KUKA KRL program: MyProgram_083().src

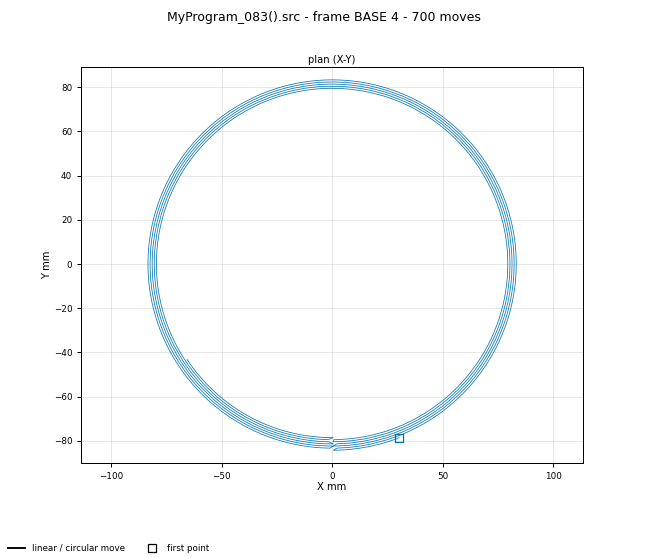
[picture p0: tool path of MyProgram_083().src in frame BASE 4, 700 of 700 moves have a stored position in this frame; points joined in program order, loops and branches not executed]
&ACCESS RVP
&REL 1
&PARAM TEMPLATE = C:\KRC\Roboter\Template\vorgabe
&PARAM EDITMASK = *
DEF MyProgram_083()
; ---- Setting reference (Base) ----
$BASE = BASE_DATA[4]

; --------------------------
; ---- Setting tool (TCP) ----
$TOOL = TOOL_DATA[3]
; --------------------------

$VEL.CP = VEL_APROX_PRINT
Startdeposition()
$VEL.CP = VEL_PRINT
LIN {X 30.3148,Y -78.5882,Z 83,A -74.2306,B 24.9241,C -2.0111,E1 25.0564,E2 519.1273} C_DIS
LIN {X 27.4017,Y -79.6507,Z 83,A -76.334,B 24.9244,C -2.0086,E1 25.0508,E2 521.2324} C_DIS
LIN {X 24.5836,Y -80.5643,Z 83,A -78.3586,B 24.9246,C -2.0059,E1 25.0454,E2 523.2596} C_DIS
LIN {X 21.4679,Y -81.4507,Z 83,A -80.5864,B 24.9248,C -2.0028,E1 25.0394,E2 525.4912} C_DIS
LIN {X 18.4554,Y -82.1857,Z 83,A -82.6471,B 24.9248,C -2.0023,E1 25.0338,E2 527.5502} C_DIS
LIN {X 15.4179,Y -82.8093,Z 83,A -84.7526,B 24.9249,C -2.0007,E1 25.028,E2 529.6571} C_DIS
LIN {X 12.3595,Y -83.3207,Z 83,A -86.9027,B 24.9252,C -1.9979,E1 25.0221,E2 531.8118} C_DIS
LIN {X 9.2843,Y -83.7191,Z 83,A -88.9651,B 24.9252,C -1.9981,E1 25.0164,E2 533.8722} C_DIS
LIN {X 6.1965,Y -84.0041,Z 83,A -91.0724,B 24.9252,C -1.9971,E1 25.0105,E2 535.9806} C_DIS
LIN {X 3.1004,Y -84.1753,Z 83,A -93.1799,B 24.9252,C -1.9963,E1 25.0046,E2 538.0892} C_DIS
LIN {X 0.5591,Y -84.2264,Z 83,A -94.1723,B 24.9236,C -2.0186,E1 25.002,E2 539.0288} C_DIS
Enddeposition()
LIN {X 0.5591,Y -84.2264,Z 83,A -94.1723,B 24.9236,C -2.0186,E1 25.002,E2 539.0288} C_DIS
Startdeposition()
$VEL.CP = VEL_PRINT
LIN {X 2.2766,Y -83.2483,Z 83,A -92.7209,B 24.9217,C -2.0436,E1 25.0063,E2 537.5182} C_DIS
LIN {X 5.5272,Y -83.0953,Z 83,A -90.5271,B 24.9217,C -2.0432,E1 25.0123,E2 535.3263} C_DIS
LIN {X 8.4362,Y -82.8508,Z 83,A -88.4909,B 24.9216,C -2.0451,E1 25.018,E2 533.2867} C_DIS
LIN {X 11.6914,Y -82.4542,Z 83,A -86.2486,B 24.9215,C -2.0461,E1 25.0242,E2 531.0439} C_DIS
LIN {X 14.5797,Y -81.9929,Z 83,A -84.2439,B 24.9214,C -2.0474,E1 25.0297,E2 529.0382} C_DIS
LIN {X 17.6429,Y -81.3887,Z 83,A -81.6481,B 24.9202,C -2.0634,E1 25.0369,E2 526.4078} C_DIS
LIN {X 24.7884,Y -79.5043,Z 83,A -76.0551,B 24.9185,C -2.0853,E1 25.052,E2 520.7724} C_DIS
LIN {X 29.127,Y -78.0202,Z 83,A -73.8096,B 24.9204,C -2.0602,E1 25.0578,E2 518.5911} C_DIS
LIN {X 32.2733,Y -76.7712,Z 83,A -71.5414,B 24.9204,C -2.0616,E1 25.0636,E2 516.3248} C_DIS
LIN {X 35.3444,Y -75.4069,Z 83,A -69.0733,B 24.9196,C -2.0701,E1 25.0699,E2 513.8426} C_DIS
LIN {X 38.5141,Y -73.8387,Z 83,A -66.2682,B 24.9184,C -2.0862,E1 25.077,E2 511.0072} C_DIS
LIN {X 41.3644,Y -72.2799,Z 83,A -64.0651,B 24.9181,C -2.0892,E1 25.0823,E2 508.8037} C_DIS
LIN {X 45.2001,Y -69.9456,Z 83,A -61.4311,B 24.9189,C -2.0802,E1 25.0885,E2 506.1994} C_DIS
LIN {X 47.8938,Y -68.1304,Z 83,A -59.266,B 24.9187,C -2.0823,E1 25.0934,E2 504.0366} C_DIS
LIN {X 50.4528,Y -66.258,Z 83,A -57.0629,B 24.9183,C -2.0876,E1 25.0984,E2 501.829} C_DIS
LIN {X 53.1162,Y -64.141,Z 83,A -54.8286,B 24.9181,C -2.0893,E1 25.1032,E2 499.5992} C_DIS
LIN {X 56.0538,Y -61.5911,Z 83,A -51.8123,B 24.9168,C -2.1066,E1 25.1096,E2 496.554} C_DIS
LIN {X 59.1004,Y -58.6733,Z 83,A -49.1949,B 24.917,C -2.1041,E1 25.1147,E2 493.9533} C_DIS
LIN {X 61.4699,Y -56.1859,Z 83,A -47.1294,B 24.9173,C -2.1002,E1 25.1186,E2 491.9062} C_DIS
LIN {X 64.0988,Y -53.1669,Z 83,A -44.0567,B 24.9159,C -2.1178,E1 25.1243,E2 488.8059} C_DIS
LIN {X 67.1499,Y -49.2572,Z 83,A -40.7875,B 24.9155,C -2.1221,E1 25.1298,E2 485.5419} C_DIS
LIN {X 68.7353,Y -47.0206,Z 83,A -38.365,B 24.9137,C -2.1453,E1 25.1337,E2 483.0767} C_DIS
LIN {X 71.2353,Y -43.1385,Z 83,A -35.7477,B 24.9145,C -2.1355,E1 25.1375,E2 480.4957} C_DIS
LIN {X 72.5407,Y -40.9065,Z 83,A -33.8555,B 24.9138,C -2.1444,E1 25.1402,E2 478.5923} C_DIS
LIN {X 74.1839,Y -37.8435,Z 83,A -31.5501,B 24.9134,C -2.1485,E1 25.1431,E2 476.2894} C_DIS
LIN {X 75.7192,Y -34.673,Z 83,A -29.1809,B 24.913,C -2.1539,E1 25.146,E2 473.9202} C_DIS
LIN {X 78.0639,Y -29.0114,Z 83,A -24.9527,B 24.9119,C -2.1671,E1 25.1504,E2 469.6842} C_DIS
LIN {X 79.3994,Y -25.1265,Z 83,A -22.1584,B 24.9113,C -2.1748,E1 25.1528,E2 466.8876} C_DIS
LIN {X 80.2886,Y -22.1198,Z 83,A -19.9737,B 24.9107,C -2.1825,E1 25.1545,E2 464.6972} C_DIS
LIN {X 81.1089,Y -18.8877,Z 83,A -17.759,B 24.9103,C -2.187,E1 25.156,E2 462.4846} C_DIS
LIN {X 81.8011,Y -15.6197,Z 83,A -15.3853,B 24.9095,C -2.1969,E1 25.1573,E2 460.1016} C_DIS
LIN {X 82.4143,Y -11.9722,Z 83,A -13.1383,B 24.9096,C -2.1949,E1 25.1583,E2 457.8722} C_DIS
LIN {X 82.7817,Y -9.0968,Z 83,A -10.9181,B 24.9085,C -2.2089,E1 25.159,E2 455.6322} C_DIS
LIN {X 83.0508,Y -6.1767,Z 83,A -9.0557,B 24.9084,C -2.2101,E1 25.1594,E2 453.778} C_DIS
LIN {X 83.1967,Y -3.7006,Z 83,A -7.1515,B 24.9074,C -2.2223,E1 25.1597,E2 451.8564} C_DIS
LIN {X 83.2798,Y 0.1338,Z 83,A -4.6895,B 24.9072,C -2.2247,E1 25.1597,E2 449.4032} C_DIS
LIN {X 83.2317,Y 2.8163,Z 83,A -2.9547,B 24.907,C -2.2269,E1 25.1597,E2 447.6737} C_DIS
LIN {X 83.0758,Y 5.8158,Z 83,A -0.6903,B 24.9059,C -2.2401,E1 25.1593,E2 445.3915} C_DIS
LIN {X 82.796,Y 8.96,Z 83,A 1.5055,B 24.9052,C -2.2477,E1 25.1586,E2 443.1907} C_DIS
LIN {X 82.3293,Y 12.5416,Z 83,A 3.8863,B 24.9049,C -2.252,E1 25.1577,E2 440.8138} C_DIS
LIN {X 81.7324,Y 15.9765,Z 83,A 6.3167,B 24.9041,C -2.2605,E1 25.1565,E2 438.3776} C_DIS
LIN {X 81.047,Y 19.1557,Z 83,A 8.3166,B 24.9042,C -2.2594,E1 25.1553,E2 436.3919} C_DIS
LIN {X 79.9547,Y 23.2977,Z 83,A 11.4453,B 24.903,C -2.2744,E1 25.153,E2 433.2459} C_DIS
LIN {X 78.9726,Y 26.4336,Z 83,A 13.6144,B 24.9026,C -2.278,E1 25.1511,E2 431.0804} C_DIS
LIN {X 78.1039,Y 28.9017,Z 83,A 15.9195,B 24.9007,C -2.3002,E1 25.1488,E2 428.7359} C_DIS
LIN {X 76.3834,Y 33.1808,Z 83,A 18.5771,B 24.9014,C -2.2921,E1 25.146,E2 426.112} C_DIS
LIN {X 74.9893,Y 36.2217,Z 83,A 20.8163,B 24.9011,C -2.2964,E1 25.1433,E2 423.8746} C_DIS
LIN {X 73.5484,Y 39.0652,Z 83,A 23.1175,B 24.9002,C -2.306,E1 25.1404,E2 421.563} C_DIS
LIN {X 72.3086,Y 41.3145,Z 83,A 24.9996,B 24.8995,C -2.3145,E1 25.1378,E2 419.6705} C_DIS
LIN {X 70.4163,Y 44.4645,Z 83,A 27.2243,B 24.8998,C -2.3111,E1 25.1345,E2 417.4651} C_DIS
LIN {X 68.659,Y 47.1334,Z 83,A 29.3239,B 24.8996,C -2.3134,E1 25.1313,E2 415.3705} C_DIS
LIN {X 66.949,Y 49.5316,Z 83,A 31.5565,B 24.8986,C -2.3252,E1 25.1276,E2 413.121} C_DIS
LIN {X 65.0896,Y 51.9507,Z 83,A 33.6147,B 24.8982,C -2.3288,E1 25.124,E2 411.0638} C_DIS
LIN {X 63.2176,Y 54.2123,Z 83,A 35.6181,B 24.8979,C -2.333,E1 25.1204,E2 409.0597} C_DIS
LIN {X 60.497,Y 57.2324,Z 83,A 38.4466,B 24.8972,C -2.3402,E1 25.1151,E2 406.2267} C_DIS
LIN {X 58.1763,Y 59.5914,Z 83,A 40.7466,B 24.8968,C -2.3457,E1 25.1105,E2 403.9233} C_DIS
LIN {X 56.3761,Y 61.2954,Z 83,A 42.6082,B 24.896,C -2.3542,E1 25.1067,E2 402.0492} C_DIS
LIN {X 53.5749,Y 63.7598,Z 83,A 45.0221,B 24.896,C -2.3542,E1 25.1016,E2 399.6447} C_DIS
LIN {X 50.8443,Y 65.9563,Z 83,A 47.0753,B 24.8966,C -2.3472,E1 25.0971,E2 397.6158} C_DIS
LIN {X 48.675,Y 67.5741,Z 83,A 49.1394,B 24.8958,C -2.3568,E1 25.0925,E2 395.5362} C_DIS
LIN {X 46.1454,Y 69.3261,Z 83,A 51.7586,B 24.894,C -2.3762,E1 25.0863,E2 392.8798} C_DIS
LIN {X 41.7622,Y 72.0513,Z 83,A 54.8615,B 24.8948,C -2.3672,E1 25.079,E2 389.8078} C_DIS
LIN {X 38.8786,Y 73.6467,Z 83,A 57.1378,B 24.8945,C -2.3706,E1 25.0734,E2 387.5302} C_DIS
LIN {X 35.9344,Y 75.1273,Z 83,A 59.3109,B 24.8945,C -2.3704,E1 25.0679,E2 385.3633} C_DIS
LIN {X 33.2525,Y 76.3521,Z 83,A 61.146,B 24.8949,C -2.3666,E1 25.0633,E2 383.5416} C_DIS
LIN {X 29.1509,Y 78.0111,Z 83,A 64.9693,B 24.8925,C -2.3939,E1 25.0532,E2 379.6623} C_DIS
LIN {X 26.0378,Y 79.1049,Z 83,A 66.6073,B 24.8941,C -2.3761,E1 25.049,E2 378.0695} C_DIS
LIN {X 24.074,Y 79.7244,Z 83,A 68.1871,B 24.8935,C -2.3822,E1 25.0447,E2 376.4781} C_DIS
LIN {X 20.7113,Y 80.6624,Z 83,A 70.3301,B 24.8941,C -2.3758,E1 25.039,E2 374.3537} C_DIS
LIN {X 18.1998,Y 81.2672,Z 83,A 72.3695,B 24.8933,C -2.3847,E1 25.0334,E2 372.2959} C_DIS
LIN {X 14.9781,Y 81.9212,Z 83,A 74.5372,B 24.8935,C -2.3828,E1 25.0275,E2 370.1353} C_DIS
LIN {X 12.2266,Y 82.3779,Z 83,A 76.2737,B 24.8939,C -2.3778,E1 25.0227,E2 368.4123} C_DIS
LIN {X 9.7923,Y 82.7013,Z 83,A 78.135,B 24.8934,C -2.3834,E1 25.0175,E2 366.5393} C_DIS
LIN {X 6.4728,Y 83.0271,Z 83,A 80.4499,B 24.8934,C -2.3842,E1 25.0111,E2 364.2238} C_DIS
LIN {X 3.2103,Y 83.2178,Z 83,A 82.8056,B 24.8931,C -2.3873,E1 25.0045,E2 361.8615} C_DIS
LIN {X -0.433,Y 83.2778,Z 83,A 85.1471,B 24.8935,C -2.3819,E1 24.998,E2 359.5329} C_DIS
LIN {X -3.6284,Y 83.1998,Z 83,A 87.3137,B 24.8937,C -2.3803,E1 24.992,E2 357.3698} C_DIS
LIN {X -6.4631,Y 83.0279,Z 83,A 89.3062,B 24.8937,C -2.3806,E1 24.9864,E2 355.3758} C_DIS
LIN {X -10.1051,Y 82.6646,Z 83,A 91.8731,B 24.8937,C -2.3806,E1 24.9793,E2 352.8072} C_DIS
LIN {X -13.5154,Y 82.1752,Z 83,A 94.2123,B 24.8939,C -2.3782,E1 24.9728,E2 350.4719} C_DIS
LIN {X -16.3634,Y 81.6564,Z 83,A 96.287,B 24.8938,C -2.379,E1 24.9671,E2 348.3929} C_DIS
LIN {X -19.702,Y 80.9148,Z 83,A 98.5118,B 24.8943,C -2.3732,E1 24.9611,E2 346.1791} C_DIS
LIN {X -22.4154,Y 80.2061,Z 83,A 100.4183,B 24.8946,C -2.3705,E1 24.956,E2 344.2759} C_DIS
LIN {X -24.918,Y 79.4641,Z 83,A 102.3404,B 24.8944,C -2.3722,E1 24.9508,E2 342.3467} C_DIS
LIN {X -27.7638,Y 78.5149,Z 83,A 104.7794,B 24.8937,C -2.3804,E1 24.9443,E2 339.8832} C_DIS
LIN {X -31.8944,Y 76.9307,Z 83,A 107.4713,B 24.8949,C -2.3662,E1 24.9374,E2 337.2195} C_DIS
LIN {X -34.8305,Y 75.6461,Z 83,A 109.7266,B 24.8951,C -2.3643,E1 24.9317,E2 334.963} C_DIS
LIN {X -41.0642,Y 72.4518,Z 83,A 114.2822,B 24.8965,C -2.3489,E1 24.9205,E2 330.4317} C_DIS
LIN {X -43.5772,Y 70.9687,Z 83,A 116.6283,B 24.896,C -2.3548,E1 24.9148,E2 328.0644} C_DIS
LIN {X -46.1606,Y 69.3161,Z 83,A 118.8803,B 24.896,C -2.3548,E1 24.9095,E2 325.8051} C_DIS
LIN {X -49.3998,Y 67.0455,Z 83,A 121.4238,B 24.8969,C -2.3442,E1 24.9038,E2 323.2778} C_DIS
LIN {X -52.0211,Y 65.0339,Z 83,A 123.4956,B 24.8978,C -2.3338,E1 24.8993,E2 321.2231} C_DIS
LIN {X -54.4202,Y 63.04,Z 83,A 126.0988,B 24.8971,C -2.3417,E1 24.8937,E2 318.591} C_DIS
LIN {X -57.2714,Y 60.4604,Z 83,A 128.4357,B 24.8984,C -2.3271,E1 24.8889,E2 316.2794} C_DIS
LIN {X -59.3395,Y 58.4313,Z 83,A 130.5413,B 24.8985,C -2.3254,E1 24.8848,E2 314.169} C_DIS
LIN {X -61.8347,Y 55.7848,Z 83,A 132.9601,B 24.8993,C -2.3169,E1 24.8802,E2 311.7598} C_DIS
LIN {X -64.2217,Y 53.0191,Z 83,A 135.5053,B 24.8998,C -2.3114,E1 24.8756,E2 309.2162} C_DIS
LIN {X -66.1385,Y 50.6079,Z 83,A 137.4999,B 24.9005,C -2.3024,E1 24.8722,E2 307.2336} C_DIS
LIN {X -68.0525,Y 48.0045,Z 83,A 139.9954,B 24.9005,C -2.3038,E1 24.8681,E2 304.7225} C_DIS
LIN {X -71.4518,Y 42.7801,Z 83,A 143.9677,B 24.9022,C -2.2832,E1 24.8622,E2 300.7793} C_DIS
LIN {X -73.1359,Y 39.8313,Z 83,A 146.5293,B 24.9022,C -2.2826,E1 24.8587,E2 298.2058} C_DIS
LIN {X -74.6288,Y 36.9583,Z 83,A 148.8382,B 24.9026,C -2.2783,E1 24.8558,E2 295.8948} C_DIS
LIN {X -76.0363,Y 33.9695,Z 83,A 151.2402,B 24.9029,C -2.275,E1 24.853,E2 293.4876} C_DIS
LIN {X -77.4282,Y 30.6645,Z 83,A 153.607,B 24.9038,C -2.2648,E1 24.8505,E2 291.1318} C_DIS
LIN {X -78.3743,Y 28.1604,Z 83,A 155.2561,B 24.9047,C -2.254,E1 24.8489,E2 289.4992} C_DIS
LIN {X -79.7646,Y 23.9384,Z 83,A 158.5508,B 24.905,C -2.2508,E1 24.8461,E2 286.1931} C_DIS
LIN {X -80.7118,Y 20.5192,Z 83,A 160.9934,B 24.9056,C -2.2432,E1 24.8443,E2 283.7545} C_DIS
LIN {X -81.2535,Y 18.2619,Z 83,A 163.0357,B 24.905,C -2.2502,E1 24.8431,E2 281.6836} C_DIS
LIN {X -82.1577,Y 13.62,Z 83,A 165.639,B 24.9074,C -2.2224,E1 24.8418,E2 279.1312} C_DIS
LIN {X -82.6677,Y 10.0792,Z 83,A 168.3253,B 24.9075,C -2.2206,E1 24.8408,E2 276.4333} C_DIS
LIN {X -82.9964,Y 6.8574,Z 83,A 170.4206,B 24.9084,C -2.2099,E1 24.8402,E2 274.3509} C_DIS
LIN {X -83.1884,Y 3.8947,Z 83,A 172.6479,B 24.9085,C -2.2083,E1 24.8399,E2 272.1139} C_DIS
LIN {X -83.2762,Y 0.7426,Z 83,A 174.7922,B 24.9092,C -2.2007,E1 24.8398,E2 269.9748} C_DIS
LIN {X -83.2493,Y -2.2433,Z 83,A 176.8695,B 24.9096,C -2.1948,E1 24.8398,E2 267.8991} C_DIS
LIN {X -83.1174,Y -5.2015,Z 83,A 178.9156,B 24.9102,C -2.1886,E1 24.8402,E2 265.8556} C_DIS
LIN {X -82.869,Y -8.263,Z 83,A -178.9161,B 24.9106,C -2.1834,E1 24.8407,E2 263.6867} C_DIS
LIN {X -82.5154,Y -11.2599,Z 83,A -176.8353,B 24.9111,C -2.177,E1 24.8415,E2 261.6086} C_DIS
LIN {X -82.0089,Y -14.491,Z 83,A -174.0318,B 24.9104,C -2.1851,E1 24.8428,E2 258.7694} C_DIS
LIN {X -81.3812,Y -17.6772,Z 83,A -172.376,B 24.9123,C -2.1625,E1 24.8438,E2 257.1577} C_DIS
LIN {X -80.806,Y -20.148,Z 83,A -170.2993,B 24.912,C -2.1661,E1 24.8452,E2 255.0601} C_DIS
LIN {X -79.7539,Y -23.9746,Z 83,A -167.8923,B 24.9134,C -2.1492,E1 24.847,E2 252.6797} C_DIS
LIN {X -78.8305,Y -26.8552,Z 83,A -165.8053,B 24.9139,C -2.1432,E1 24.8488,E2 250.5951} C_DIS
LIN {X -77.9352,Y -29.3513,Z 83,A -163.8576,B 24.914,C -2.1412,E1 24.8507,E2 248.641} C_DIS
LIN {X -76.8139,Y -32.172,Z 83,A -161.7124,B 24.9144,C -2.1368,E1 24.853,E2 246.4945} C_DIS
LIN {X -75.485,Y -35.1767,Z 83,A -159.5329,B 24.9151,C -2.1282,E1 24.8555,E2 244.3234} C_DIS
LIN {X -73.9824,Y -38.2378,Z 83,A -157.1587,B 24.9155,C -2.1225,E1 24.8585,E2 241.9501} C_DIS
LIN {X -72.4839,Y -41.0083,Z 83,A -154.8521,B 24.9157,C -2.1206,E1 24.8616,E2 239.6361} C_DIS
LIN {X -70.6438,Y -44.1002,Z 83,A -152.5429,B 24.9165,C -2.1095,E1 24.8649,E2 237.3413} C_DIS
LIN {X -69.2182,Y -46.3077,Z 83,A -150.0661,B 24.9154,C -2.1235,E1 24.8689,E2 234.8187} C_DIS
LIN {X -67.277,Y -49.0836,Z 83,A -148.293,B 24.9171,C -2.1023,E1 24.8717,E2 233.0878} C_DIS
LIN {X -65.2096,Y -51.7989,Z 83,A -146.2559,B 24.9182,C -2.088,E1 24.8751,E2 231.075} C_DIS
LIN {X -63.0232,Y -54.4395,Z 83,A -143.4942,B 24.9178,C -2.0938,E1 24.8801,E2 228.2867} C_DIS
LIN {X -60.8121,Y -56.8974,Z 83,A -141.3418,B 24.9184,C -2.0854,E1 24.8842,E2 226.1449} C_DIS
LIN {X -58.9873,Y -58.7879,Z 83,A -138.93,B 24.9174,C -2.0987,E1 24.889,E2 223.6911} C_DIS
LIN {X -56.6005,Y -61.0895,Z 83,A -137.1338,B 24.9188,C -2.0803,E1 24.8926,E2 221.9315} C_DIS
LIN {X -54.085,Y -63.3261,Z 83,A -134.6178,B 24.9188,C -2.0816,E1 24.8979,E2 219.4026} C_DIS
LIN {X -50.8394,Y -65.9601,Z 83,A -131.9262,B 24.9196,C -2.0711,E1 24.9038,E2 216.726} C_DIS
LIN {X -48.6875,Y -67.5652,Z 83,A -129.5874,B 24.9187,C -2.0821,E1 24.9092,E2 214.3527} C_DIS
LIN {X -46.0328,Y -69.4004,Z 83,A -127.8872,B 24.9201,C -2.0636,E1 24.913,E2 212.691} C_DIS
LIN {X -42.9611,Y -71.3431,Z 83,A -125.3297,B 24.9203,C -2.0615,E1 24.9191,E2 210.1304} C_DIS
LIN {X -40.114,Y -72.9826,Z 83,A -123.2403,B 24.9209,C -2.0535,E1 24.9242,E2 208.0541} C_DIS
LIN {X -37.7618,Y -74.2256,Z 83,A -121.4189,B 24.9211,C -2.0509,E1 24.9287,E2 206.2338} C_DIS
LIN {X -35.3141,Y -75.421,Z 83,A -118.7338,B 24.9194,C -2.0726,E1 24.9356,E2 203.4904} C_DIS
LIN {X -31.9021,Y -76.9276,Z 83,A -116.0869,B 24.9194,C -2.0724,E1 24.9424,E2 200.838} C_DIS
LIN {X -28.2936,Y -78.3257,Z 83,A -114.32,B 24.9217,C -2.0434,E1 24.9469,E2 199.1363} C_DIS
LIN {X -25.3736,Y -79.3198,Z 83,A -111.9912,B 24.9214,C -2.0479,E1 24.9531,E2 196.7926} C_DIS
LIN {X -22.809,Y -80.0946,Z 83,A -110.2382,B 24.9217,C -2.044,E1 24.9578,E2 195.0461} C_DIS
LIN {X -19.6726,Y -80.922,Z 83,A -107.9499,B 24.9217,C -2.0444,E1 24.964,E2 192.7535} C_DIS
LIN {X -16.8864,Y -81.5491,Z 83,A -106.0101,B 24.9217,C -2.0428,E1 24.9693,E2 190.8152} C_DIS
LIN {X -13.5662,Y -82.1667,Z 83,A -103.7836,B 24.922,C -2.0391,E1 24.9754,E2 188.5951} C_DIS
LIN {X -10.5031,Y -82.6142,Z 83,A -101.4942,B 24.9217,C -2.0435,E1 24.9818,E2 186.2935} C_DIS
LIN {X -7.1182,Y -82.9756,Z 83,A -99.121,B 24.9217,C -2.0442,E1 24.9884,E2 183.9173} C_DIS
LIN {X -4.5308,Y -83.1556,Z 83,A -97.373,B 24.9217,C -2.0432,E1 24.9932,E2 182.1712} C_DIS
LIN {X -1.0027,Y -83.2741,Z 83,A -94.9241,B 24.9217,C -2.0442,E1 25.0001,E2 179.7197} C_DIS
LIN {X -1.0027,Y -83.2741,Z 83,A -94.9241,B 24.9217,C -2.0442,E1 25.0001,E2 179.7197} C_DIS
Enddeposition()
LIN {X 0.5504,Y -82.3231,Z 83,A -94.2468,B 24.9213,C -2.049,E1 25.002,E2 179.031} C_DIS
Startdeposition()
$VEL.CP = VEL_PRINT
LIN {X -1.5524,Y -82.3124,Z 83,A -96.6682,B 24.9235,C -2.0201,E1 24.9951,E2 181.5212} C_DIS
LIN {X -5.6861,Y -82.1306,Z 83,A -99.1832,B 24.9227,C -2.0307,E1 24.9881,E2 184.0117} C_DIS
LIN {X -8.7147,Y -81.8646,Z 83,A -101.4384,B 24.923,C -2.0267,E1 24.9818,E2 186.2775} C_DIS
LIN {X -11.9249,Y -81.4596,Z 83,A -103.7765,B 24.9231,C -2.0247,E1 24.9753,E2 188.6223} C_DIS
LIN {X -15.5144,Y -80.852,Z 83,A -106.1545,B 24.9227,C -2.0301,E1 24.9688,E2 190.99} C_DIS
LIN {X -18.5189,Y -80.2172,Z 83,A -108.3547,B 24.9227,C -2.0292,E1 24.9628,E2 193.1948} C_DIS
LIN {X -22.5796,Y -79.1702,Z 83,A -110.9842,B 24.922,C -2.0393,E1 24.9558,E2 195.8044} C_DIS
LIN {X -24.8256,Y -78.4957,Z 83,A -113.2233,B 24.9233,C -2.023,E1 24.9497,E2 198.086} C_DIS
LIN {X -28.7698,Y -77.1376,Z 83,A -116.3221,B 24.9235,C -2.02,E1 24.9415,E2 201.1981} C_DIS
LIN {X -34.6143,Y -74.6968,Z 83,A -120.2039,B 24.922,C -2.0396,E1 24.9317,E2 205.0426} C_DIS
LIN {X -37.6746,Y -73.2013,Z 83,A -122.7566,B 24.9222,C -2.0374,E1 24.9253,E2 207.6075} C_DIS
LIN {X -40.8894,Y -71.455,Z 83,A -125.1525,B 24.9216,C -2.045,E1 24.9194,E2 209.992} C_DIS
LIN {X -43.7124,Y -69.7638,Z 83,A -127.7428,B 24.922,C -2.0401,E1 24.9132,E2 212.6022} C_DIS
LIN {X -48.0318,Y -66.8637,Z 83,A -131.0831,B 24.9209,C -2.0537,E1 24.9056,E2 215.9213} C_DIS
LIN {X -50.4597,Y -65.051,Z 83,A -133.24,B 24.9207,C -2.0561,E1 24.9008,E2 218.0804} C_DIS
LIN {X -53.9999,Y -62.1434,Z 83,A -136.1063,B 24.9196,C -2.0709,E1 24.8947,E2 220.9224} C_DIS
LIN {X -56.6894,Y -59.701,Z 83,A -139.5018,B 24.921,C -2.0523,E1 24.8876,E2 224.3759} C_DIS
LIN {X -58.9888,Y -57.4303,Z 83,A -141.2543,B 24.9196,C -2.0705,E1 24.8843,E2 226.0926} C_DIS
LIN {X -61.1234,Y -55.1523,Z 83,A -144.227,B 24.9209,C -2.0538,E1 24.8786,E2 229.1183} C_DIS
LIN {X -63.782,Y -52.0545,Z 83,A -146.3247,B 24.9188,C -2.0802,E1 24.875,E2 231.1626} C_DIS
LIN {X -66.5611,Y -48.4501,Z 83,A -149.7864,B 24.9188,C -2.08,E1 24.8691,E2 234.6415} C_DIS
LIN {X -69.0207,Y -44.879,Z 83,A -152.4967,B 24.9176,C -2.0958,E1 24.865,E2 237.3277} C_DIS
LIN {X -70.5517,Y -42.4305,Z 83,A -155.1104,B 24.9185,C -2.0851,E1 24.8611,E2 239.9804} C_DIS
LIN {X -72.2473,Y -39.4733,Z 83,A -156.9169,B 24.9168,C -2.1064,E1 24.8587,E2 241.7455} C_DIS
LIN {X -73.8018,Y -36.4834,Z 83,A -159.2444,B 24.9162,C -2.1133,E1 24.8558,E2 244.0691} C_DIS
LIN {X -75.8072,Y -32.1097,Z 83,A -162.5765,B 24.9155,C -2.1231,E1 24.852,E2 247.3959} C_DIS
LIN {X -76.9221,Y -29.3391,Z 83,A -164.668,B 24.915,C -2.1288,E1 24.8499,E2 249.4857} C_DIS
LIN {X -77.9197,Y -26.5773,Z 83,A -166.7483,B 24.9146,C -2.1338,E1 24.8479,E2 251.5658} C_DIS
LIN {X -78.9025,Y -23.4978,Z 83,A -169.0526,B 24.9142,C -2.1391,E1 24.846,E2 253.8707} C_DIS
LIN {X -80.1273,Y -18.9078,Z 83,A -172.4738,B 24.9136,C -2.1461,E1 24.8437,E2 257.2951} C_DIS
LIN {X -81.1733,Y -13.7358,Z 83,A -175.6492,B 24.9116,C -2.1704,E1 24.842,E2 260.4312} C_DIS
LIN {X -81.5066,Y -11.594,Z 83,A -177.5733,B 24.9121,C -2.1643,E1 24.8412,E2 262.3815} C_DIS
LIN {X -82.0324,Y -6.972,Z 83,A 178.7589,B 24.9122,C -2.1633,E1 24.8402,E2 266.0735} C_DIS
LIN {X -82.2721,Y -3.0466,Z 83,A 176.3153,B 24.9109,C -2.1796,E1 24.8398,E2 268.4931} C_DIS
LIN {X -82.3268,Y 0.3626,Z 83,A 173.6639,B 24.9109,C -2.18,E1 24.8398,E2 271.1595} C_DIS
LIN {X -82.0421,Y 6.8502,Z 83,A 169.7779,B 24.9083,C -2.2108,E1 24.8404,E2 274.9953} C_DIS
LIN {X -81.6591,Y 10.4669,Z 83,A 166.5866,B 24.9091,C -2.2018,E1 24.8414,E2 278.2273} C_DIS
LIN {X -81.2236,Y 13.4345,Z 83,A 164.049,B 24.9095,C -2.1968,E1 24.8426,E2 280.7917} C_DIS
LIN {X -80.5008,Y 17.243,Z 83,A 162.0067,B 24.9074,C -2.2222,E1 24.8437,E2 282.7855} C_DIS
LIN {X -79.9755,Y 19.5361,Z 83,A 159.576,B 24.9086,C -2.207,E1 24.8454,E2 285.2667} C_DIS
LIN {X -78.8665,Y 23.6193,Z 83,A 157.1283,B 24.9068,C -2.2288,E1 24.8473,E2 287.6764} C_DIS
LIN {X -77.4401,Y 27.9437,Z 83,A 154.6172,B 24.9046,C -2.2557,E1 24.8495,E2 290.1378} C_DIS
LIN {X -76.529,Y 30.3501,Z 83,A 152.4182,B 24.905,C -2.2505,E1 24.8517,E2 292.3615} C_DIS
LIN {X -74.1199,Y 35.8333,Z 83,A 148.4322,B 24.9035,C -2.2677,E1 24.8563,E2 296.3283} C_DIS
LIN {X -71.2191,Y 41.3001,Z 83,A 144.1422,B 24.9024,C -2.2806,E1 24.862,E2 300.6102} C_DIS
LIN {X -70.2138,Y 42.9864,Z 83,A 141.9782,B 24.9039,C -2.2636,E1 24.8652,E2 302.8258} C_DIS
LIN {X -68.3701,Y 45.8628,Z 83,A 140.1448,B 24.9021,C -2.2844,E1 24.868,E2 304.6189} C_DIS
LIN {X -65.4603,Y 49.9285,Z 83,A 136.7915,B 24.901,C -2.297,E1 24.8735,E2 307.9581} C_DIS
LIN {X -62.0296,Y 54.1301,Z 83,A 133.0235,B 24.9001,C -2.3069,E1 24.8802,E2 311.7199} C_DIS
LIN {X -59.2782,Y 57.13,Z 83,A 130.55,B 24.8987,C -2.3235,E1 24.8848,E2 314.1648} C_DIS
LIN {X -57.8082,Y 58.617,Z 83,A 128.5469,B 24.8997,C -2.3124,E1 24.8888,E2 316.2029} C_DIS
LIN {X -54.1458,Y 62.016,Z 83,A 125.3768,B 24.8983,C -2.3286,E1 24.8953,E2 319.3472} C_DIS
LIN {X -50.9579,Y 64.6611,Z 83,A 122.3567,B 24.898,C -2.3311,E1 24.9018,E2 322.3727} C_DIS
LIN {X -48.8772,Y 66.2484,Z 83,A 119.525,B 24.9001,C -2.3078,E1 24.9083,E2 325.2699} C_DIS
LIN {X -45.5242,Y 68.5956,Z 83,A 117.8431,B 24.8968,C -2.3447,E1 24.912,E2 326.8695} C_DIS
LIN {X -42.0842,Y 70.7581,Z 83,A 114.7218,B 24.8971,C -2.342,E1 24.9194,E2 330.0073} C_DIS
LIN {X -38.4333,Y 72.8054,Z 83,A 111.4114,B 24.8976,C -2.3361,E1 24.9276,E2 333.3411} C_DIS
LIN {X -35.4537,Y 74.3023,Z 83,A 109.3633,B 24.8966,C -2.3472,E1 24.9327,E2 335.368} C_DIS
LIN {X -32.558,Y 75.6165,Z 83,A 107.135,B 24.8964,C -2.35,E1 24.9384,E2 337.595} C_DIS
LIN {X -27.5644,Y 77.5761,Z 83,A 103.429,B 24.8959,C -2.3557,E1 24.948,E2 341.2953} C_DIS
LIN {X -23.8211,Y 78.8061,Z 83,A 100.2076,B 24.8968,C -2.3455,E1 24.9567,E2 344.5465} C_DIS
LIN {X -19.399,Y 80.009,Z 83,A 97.4156,B 24.8955,C -2.3597,E1 24.9642,E2 347.3088} C_DIS
LIN {X -16.0884,Y 80.7412,Z 83,A 94.203,B 24.8975,C -2.3378,E1 24.9731,E2 350.5772} C_DIS
LIN {X -11.8028,Y 81.4769,Z 83,A 92.347,B 24.8943,C -2.3728,E1 24.978,E2 352.3515} C_DIS
LIN {X -7.1632,Y 82.0158,Z 83,A 89.0161,B 24.8943,C -2.3723,E1 24.9873,E2 355.6859} C_DIS
LIN {X -4.347,Y 82.2124,Z 83,A 86.8115,B 24.8949,C -2.3662,E1 24.9935,E2 357.9058} C_DIS
LIN {X 0.5328,Y 82.3253,Z 83,A 83.2747,B 24.8952,C -2.3629,E1 25.0034,E2 361.4503} C_DIS
LIN {X 3.3202,Y 82.2604,Z 83,A 81.4837,B 24.8948,C -2.3674,E1 25.0083,E2 363.2303} C_DIS
LIN {X 6.5866,Y 82.0632,Z 83,A 79.2593,B 24.8947,C -2.3689,E1 25.0145,E2 365.4501} C_DIS
LIN {X 10.5225,Y 81.6518,Z 83,A 76.3504,B 24.8951,C -2.3639,E1 25.0226,E2 368.3687} C_DIS
LIN {X 13.7049,Y 81.1784,Z 83,A 74.1891,B 24.8951,C -2.3655,E1 25.0285,E2 370.5241} C_DIS
LIN {X 16.9177,Y 80.5709,Z 83,A 71.5231,B 24.8961,C -2.353,E1 25.0359,E2 373.2164} C_DIS
LIN {X 21.5203,Y 79.4646,Z 83,A 68.4024,B 24.8958,C -2.3561,E1 25.0443,E2 376.325} C_DIS
LIN {X 25.4418,Y 78.2973,Z 83,A 65.6913,B 24.8957,C -2.358,E1 25.0515,E2 379.0266} C_DIS
LIN {X 31.7462,Y 75.9604,Z 83,A 61.5346,B 24.8947,C -2.3693,E1 25.0623,E2 383.1475} C_DIS
LIN {X 36.255,Y 73.9151,Z 83,A 57.8652,B 24.8956,C -2.3585,E1 25.0716,E2 386.8333} C_DIS
LIN {X 38.8943,Y 72.5613,Z 83,A 55.6569,B 24.8962,C -2.3515,E1 25.0771,E2 389.0522} C_DIS
LIN {X 41.8717,Y 70.8837,Z 83,A 53.2243,B 24.8967,C -2.3464,E1 25.083,E2 391.4893} C_DIS
LIN {X 45.4938,Y 68.6156,Z 83,A 50.5294,B 24.8963,C -2.3504,E1 25.0893,E2 394.166} C_DIS
LIN {X 47.6472,Y 67.1382,Z 83,A 47.8331,B 24.899,C -2.3204,E1 25.0956,E2 396.9242} C_DIS
LIN {X 50.6928,Y 64.8706,Z 83,A 45.9418,B 24.8974,C -2.3388,E1 25.0997,E2 398.765} C_DIS
LIN {X 53.0351,Y 62.9701,Z 83,A 42.9527,B 24.9001,C -2.3073,E1 25.1062,E2 401.817} C_DIS
LIN {X 56.1846,Y 60.1757,Z 83,A 40.9125,B 24.8982,C -2.329,E1 25.1103,E2 403.7975} C_DIS
LIN {X 58.4013,Y 58.0266,Z 83,A 38.7825,B 24.8986,C -2.3251,E1 25.1145,E2 405.9279} C_DIS
LIN {X 61.9206,Y 54.255,Z 83,A 35.2623,B 24.8991,C -2.3194,E1 25.1212,E2 409.4461} C_DIS
LIN {X 63.8799,Y 51.9337,Z 83,A 33.0856,B 24.8997,C -2.3125,E1 25.125,E2 411.6291} C_DIS
LIN {X 67.3106,Y 47.4055,Z 83,A 29.1432,B 24.9005,C -2.3032,E1 25.1316,E2 415.5746} C_DIS
LIN {X 69.64,Y 43.9105,Z 83,A 25.5133,B 24.903,C -2.2733,E1 25.1372,E2 419.2569} C_DIS
LIN {X 71.6242,Y 40.595,Z 83,A 23.5565,B 24.9017,C -2.2894,E1 25.1398,E2 421.1655} C_DIS
LIN {X 73.1055,Y 37.862,Z 83,A 21.3371,B 24.9023,C -2.2817,E1 25.1427,E2 423.3914} C_DIS
LIN {X 74.8291,Y 34.33,Z 83,A 18.785,B 24.9025,C -2.28,E1 25.1458,E2 425.9339} C_DIS
LIN {X 76.0477,Y 31.539,Z 83,A 16.0179,B 24.9048,C -2.2531,E1 25.1488,E2 428.7492} C_DIS
LIN {X 77.2546,Y 28.4522,Z 83,A 13.9451,B 24.9048,C -2.2539,E1 25.1508,E2 430.8086} C_DIS
LIN {X 78.349,Y 25.2821,Z 83,A 10.7448,B 24.9076,C -2.2192,E1 25.1536,E2 434.0725} C_DIS
LIN {X 79.8503,Y 20.047,Z 83,A 8.4245,B 24.9046,C -2.255,E1 25.1552,E2 436.2951} C_DIS
LIN {X 80.4835,Y 17.3262,Z 83,A 6.3022,B 24.9056,C -2.2433,E1 25.1565,E2 438.4328} C_DIS
LIN {X 81.0354,Y 14.5263,Z 83,A 4.3727,B 24.906,C -2.239,E1 25.1575,E2 440.3611} C_DIS
LIN {X 81.5472,Y 11.3083,Z 83,A 1.9681,B 24.9069,C -2.2274,E1 25.1585,E2 442.7788} C_DIS
LIN {X 81.935,Y 8.0372,Z 83,A -0.0012,B 24.9067,C -2.2307,E1 25.1591,E2 444.7286} C_DIS
LIN {X 82.1268,Y 5.7416,Z 83,A -1.7324,B 24.9074,C -2.2215,E1 25.1595,E2 446.4714} C_DIS
LIN {X 82.2747,Y 2.9706,Z 83,A -3.8226,B 24.9084,C -2.2101,E1 25.1597,E2 448.5759} C_DIS
LIN {X 82.3245,Y -0.7205,Z 83,A -6.3572,B 24.909,C -2.2031,E1 25.1597,E2 451.1121} C_DIS
LIN {X 82.2187,Y -4.2331,Z 83,A -8.6292,B 24.9091,C -2.2009,E1 25.1595,E2 453.3757} C_DIS
LIN {X 82.0138,Y -7.185,Z 83,A -10.7771,B 24.9099,C -2.1914,E1 25.159,E2 455.5332} C_DIS
LIN {X 81.5534,Y -11.2648,Z 83,A -13.2831,B 24.9097,C -2.1938,E1 25.1582,E2 458.0188} C_DIS
LIN {X 81.0227,Y -14.5968,Z 83,A -15.9377,B 24.9112,C -2.1763,E1 25.157,E2 460.6992} C_DIS
LIN {X 80.3292,Y -18.0335,Z 83,A -18.4011,B 24.9119,C -2.1678,E1 25.1555,E2 463.1684} C_DIS
LIN {X 79.5527,Y -21.1941,Z 83,A -20.5911,B 24.9122,C -2.1631,E1 25.154,E2 465.3567} C_DIS
LIN {X 78.6773,Y -24.2415,Z 83,A -22.9088,B 24.9131,C -2.1526,E1 25.1522,E2 467.686} C_DIS
LIN {X 77.6384,Y -27.3869,Z 83,A -25.1783,B 24.9136,C -2.1467,E1 25.1501,E2 469.9567} C_DIS
LIN {X 75.5519,Y -32.7064,Z 83,A -29.1683,B 24.9146,C -2.1342,E1 25.1459,E2 473.9543} C_DIS
LIN {X 74.1549,Y -35.7604,Z 83,A -31.3801,B 24.9148,C -2.1313,E1 25.1433,E2 476.1609} C_DIS
LIN {X 72.6582,Y -38.7128,Z 83,A -34.0566,B 24.9163,C -2.1124,E1 25.1398,E2 478.8678} C_DIS
LIN {X 70.2278,Y -42.9635,Z 83,A -37.1908,B 24.9163,C -2.1115,E1 25.1354,E2 481.9881} C_DIS
LIN {X 67.661,Y -46.9014,Z 83,A -40.2549,B 24.9166,C -2.1091,E1 25.1306,E2 485.0426} C_DIS
LIN {X 65.5027,Y -49.8722,Z 83,A -42.8981,B 24.9173,C -2.0994,E1 25.1262,E2 487.696} C_DIS
LIN {X 63.1426,Y -52.8283,Z 83,A -45.6448,B 24.9182,C -2.0889,E1 25.1213,E2 490.455} C_DIS
LIN {X 60.515,Y -55.8187,Z 83,A -49.2273,B 24.9207,C -2.0561,E1 25.1145,E2 494.099} C_DIS
LIN {X 57.1688,Y -59.2408,Z 83,A -51.1577,B 24.9179,C -2.0927,E1 25.1108,E2 495.9349} C_DIS
LIN {X 53.0261,Y -62.9778,Z 83,A -55.2583,B 24.9191,C -2.0767,E1 25.1022,E2 500.0569} C_DIS
LIN {X 50.2888,Y -65.1827,Z 83,A -57.934,B 24.9201,C -2.0642,E1 25.0963,E2 502.7523} C_DIS
LIN {X 47.2041,Y -67.4504,Z 83,A -60.6136,B 24.9206,C -2.0583,E1 25.0902,E2 505.4365} C_DIS
LIN {X 44.2926,Y -69.3971,Z 83,A -63.3408,B 24.9216,C -2.0445,E1 25.0838,E2 508.1874} C_DIS
LIN {X 38.6271,Y -72.7034,Z 83,A -67.1153,B 24.9203,C -2.0611,E1 25.0748,E2 511.9112} C_DIS
LIN {X 34.6749,Y -74.6686,Z 83,A -70.3057,B 24.921,C -2.0525,E1 25.0667,E2 515.1136} C_DIS
LIN {X 32.3123,Y -75.7218,Z 83,A -72.3269,B 24.9217,C -2.0429,E1 25.0615,E2 517.1526} C_DIS
LIN {X 28.9058,Y -77.0861,Z 83,A -75.1463,B 24.9226,C -2.0312,E1 25.0541,E2 519.9934} C_DIS
LIN {X 25.119,Y -78.4018,Z 83,A -77.5558,B 24.922,C -2.0395,E1 25.0478,E2 522.3788} C_DIS
LIN {X 22.2443,Y -79.2652,Z 83,A -79.8499,B 24.9227,C -2.0309,E1 25.0416,E2 524.6893} C_DIS
LIN {X 18.883,Y -80.1331,Z 83,A -82.6345,B 24.9237,C -2.0173,E1 25.034,E2 527.5021} C_DIS
LIN {X 14.1786,Y -81.0979,Z 83,A -85.4647,B 24.9227,C -2.0301,E1 25.0263,E2 530.2988} C_DIS
LIN {X 11.1465,Y -81.5702,Z 83,A -87.9139,B 24.9236,C -2.0192,E1 25.0194,E2 532.7717} C_DIS
LIN {X 7.6515,Y -81.9708,Z 83,A -90.4075,B 24.9238,C -2.0165,E1 25.0125,E2 535.2701} C_DIS
LIN {X 3.3277,Y -82.26,Z 83,A -93.1065,B 24.9231,C -2.0247,E1 25.005,E2 537.9486} C_DIS
LIN {X 0.5504,Y -82.3231,Z 83,A -94.2445,B 24.9213,C -2.0481,E1 25.002,E2 539.031} C_DIS
Enddeposition()
LIN {X 0.5504,Y -82.3231,Z 83,A -94.2445,B 24.9213,C -2.0481,E1 25.002,E2 539.031} C_DIS
Startdeposition()
$VEL.CP = VEL_PRINT
LIN {X 2.1065,Y -81.3489,Z 83,A -92.8206,B 24.9193,C -2.0747,E1 25.0062,E2 537.5442} C_DIS
LIN {X 8.1636,Y -80.9653,Z 83,A -88.9158,B 24.92,C -2.0655,E1 25.017,E2 533.6631} C_DIS
LIN {X 12.8382,Y -80.3571,Z 83,A -85.2594,B 24.919,C -2.0778,E1 25.0272,E2 529.9804} C_DIS
LIN {X 15.6467,Y -79.8572,Z 83,A -82.4389,B 24.9169,C -2.1046,E1 25.0351,E2 527.1} C_DIS
LIN {X 19.7265,Y -78.9493,Z 83,A -79.8274,B 24.9175,C -2.0971,E1 25.0421,E2 524.5099} C_DIS
LIN {X 24.6346,Y -77.5581,Z 83,A -76.9916,B 24.919,C -2.0778,E1 25.0495,E2 521.725} C_DIS
LIN {X 28.156,Y -76.3495,Z 83,A -74.4433,B 24.919,C -2.0788,E1 25.0562,E2 519.1792} C_DIS
LIN {X 31.2499,Y -75.1367,Z 83,A -71.7762,B 24.9179,C -2.0923,E1 25.0632,E2 516.4862} C_DIS
LIN {X 34.0054,Y -73.9303,Z 83,A -68.4897,B 24.9147,C -2.1325,E1 25.0718,E2 513.1128} C_DIS
LIN {X 38.7111,Y -71.5778,Z 83,A -66.4635,B 24.9184,C -2.0856,E1 25.0765,E2 511.2034} C_DIS
LIN {X 43.5339,Y -68.7529,Z 83,A -61.7057,B 24.9158,C -2.1187,E1 25.088,E2 506.382} C_DIS
LIN {X 46.9615,Y -66.4581,Z 83,A -59.2404,B 24.9165,C -2.1105,E1 25.0936,E2 503.9445} C_DIS
LIN {X 49.6061,Y -64.5071,Z 83,A -56.7231,B 24.9156,C -2.1219,E1 25.0993,E2 501.4094} C_DIS
LIN {X 52.6513,Y -62.0467,Z 83,A -54.5167,B 24.9165,C -2.1104,E1 25.104,E2 499.2386} C_DIS
LIN {X 54.9071,Y -60.0596,Z 83,A -51.9165,B 24.9149,C -2.1307,E1 25.1095,E2 496.6007} C_DIS
LIN {X 57.7737,Y -57.3075,Z 83,A -49.0226,B 24.9141,C -2.1405,E1 25.1152,E2 493.6958} C_DIS
LIN {X 60.3998,Y -54.5335,Z 83,A -46.7461,B 24.9146,C -2.1339,E1 25.1195,E2 491.445} C_DIS
LIN {X 62.4491,Y -52.1735,Z 83,A -44.2999,B 24.9135,C -2.1475,E1 25.124,E2 488.9778} C_DIS
LIN {X 64.5118,Y -49.6,Z 83,A -42.1493,B 24.9135,C -2.1481,E1 25.1277,E2 486.8358} C_DIS
LIN {X 66.9836,Y -46.2083,Z 83,A -38.1591,B 24.91,C -2.1901,E1 25.1342,E2 482.7659} C_DIS
LIN {X 69.4919,Y -42.3416,Z 83,A -36.1235,B 24.9125,C -2.1596,E1 25.1371,E2 480.8128} C_DIS
LIN {X 72.0868,Y -37.7551,Z 83,A -32.2246,B 24.9112,C -2.1764,E1 25.1424,E2 476.8944} C_DIS
LIN {X 73.5757,Y -34.7674,Z 83,A -29.4234,B 24.9094,C -2.1982,E1 25.1458,E2 474.0567} C_DIS
LIN {X 75.3369,Y -30.7618,Z 83,A -26.192,B 24.9082,C -2.2125,E1 25.1493,E2 470.8093} C_DIS
LIN {X 76.6363,Y -27.368,Z 83,A -24.5001,B 24.9099,C -2.1918,E1 25.1509,E2 469.1758} C_DIS
LIN {X 77.8235,Y -23.7811,Z 83,A -21.4295,B 24.9081,C -2.2135,E1 25.1535,E2 466.0713} C_DIS
LIN {X 78.8748,Y -20.0189,Z 83,A -18.8749,B 24.9079,C -2.2157,E1 25.1553,E2 463.5262} C_DIS
LIN {X 79.6016,Y -16.9029,Z 83,A -16.8069,B 24.9079,C -2.2168,E1 25.1566,E2 461.4678} C_DIS
LIN {X 80.4765,Y -12.0663,Z 83,A -13.5142,B 24.9074,C -2.2222,E1 25.1582,E2 458.1815} C_DIS
LIN {X 80.9821,Y -8.0031,Z 83,A -10.3222,B 24.9057,C -2.2416,E1 25.1592,E2 454.9627} C_DIS
LIN {X 81.2359,Y -4.7683,Z 83,A -8.2112,B 24.9057,C -2.2432,E1 25.1596,E2 452.8604} C_DIS
LIN {X 81.3718,Y -0.8361,Z 83,A -5.0574,B 24.9038,C -2.2646,E1 25.1598,E2 449.6748} C_DIS
LIN {X 81.3057,Y 3.3645,Z 83,A -2.4319,B 24.9039,C -2.2631,E1 25.1596,E2 447.0685} C_DIS
LIN {X 81.0653,Y 7.105,Z 83,A 0.4071,B 24.9026,C -2.278,E1 25.159,E2 444.2112} C_DIS
LIN {X 80.5144,Y 11.8103,Z 83,A 3.5504,B 24.9023,C -2.2821,E1 25.1578,E2 441.0767} C_DIS
LIN {X 79.9695,Y 15.0636,Z 83,A 5.778,B 24.9019,C -2.2862,E1 25.1567,E2 438.8524} C_DIS
LIN {X 78.9656,Y 19.6599,Z 83,A 9.7002,B 24.8993,C -2.3164,E1 25.1542,E2 434.8818} C_DIS
LIN {X 78.0778,Y 22.9302,Z 83,A 11.6493,B 24.9,C -2.3092,E1 25.1527,E2 432.9608} C_DIS
LIN {X 77.0725,Y 26.1107,Z 83,A 13.9388,B 24.8995,C -2.3142,E1 25.1507,E2 430.6723} C_DIS
LIN {X 75.2448,Y 30.9881,Z 83,A 17.4978,B 24.8989,C -2.3213,E1 25.1471,E2 427.1164} C_DIS
LIN {X 73.953,Y 33.9566,Z 83,A 20.1827,B 24.8972,C -2.3409,E1 25.144,E2 424.3998} C_DIS
LIN {X 71.9333,Y 38.0466,Z 83,A 22.8905,B 24.8978,C -2.3334,E1 25.1406,E2 421.7241} C_DIS
LIN {X 70.9374,Y 39.8731,Z 83,A 24.7668,B 24.8963,C -2.3506,E1 25.138,E2 419.8169} C_DIS
LIN {X 68.6522,Y 43.6909,Z 83,A 27.2026,B 24.8976,C -2.3363,E1 25.1345,E2 417.4272} C_DIS
LIN {X 67.0628,Y 46.0944,Z 83,A 29.2555,B 24.8971,C -2.3422,E1 25.1313,E2 415.3705} C_DIS
LIN {X 64.7314,Y 49.3151,Z 83,A 32.8514,B 24.8942,C -2.3745,E1 25.1252,E2 411.7155} C_DIS
LIN {X 62.6868,Y 51.8875,Z 83,A 34.4766,B 24.8957,C -2.358,E1 25.1224,E2 410.137} C_DIS
LIN {X 60.0111,Y 54.96,Z 83,A 37.8482,B 24.8937,C -2.3804,E1 25.1161,E2 406.7274} C_DIS
LIN {X 56.8772,Y 58.1988,Z 83,A 40.4963,B 24.8946,C -2.3704,E1 25.1109,E2 404.1141} C_DIS
LIN {X 53.6254,Y 61.2067,Z 83,A 44.2149,B 24.8923,C -2.3955,E1 25.1031,E2 400.3509} C_DIS
LIN {X 48.9494,Y 65.0069,Z 83,A 48.3462,B 24.8919,C -2.3997,E1 25.094,E2 396.2252} C_DIS
LIN {X 45.1954,Y 67.6722,Z 83,A 51.2127,B 24.8925,C -2.3933,E1 25.0875,E2 393.3836} C_DIS
LIN {X 42.647,Y 69.3063,Z 83,A 53.6791,B 24.8913,C -2.4069,E1 25.0816,E2 390.8928} C_DIS
LIN {X 38.8441,Y 71.5057,Z 83,A 56.3172,B 24.8922,C -2.3971,E1 25.0752,E2 388.2856} C_DIS
LIN {X 36.5783,Y 72.6924,Z 83,A 59.0783,B 24.8893,C -2.4289,E1 25.0682,E2 385.4566} C_DIS
LIN {X 32.652,Y 74.5372,Z 83,A 61.2132,B 24.8915,C -2.4041,E1 25.0629,E2 383.3857} C_DIS
LIN {X 28.7867,Y 76.1133,Z 83,A 64.655,B 24.8899,C -2.4223,E1 25.0538,E2 379.9084} C_DIS
LIN {X 24.3066,Y 77.6605,Z 83,A 67.3876,B 24.8913,C -2.4067,E1 25.0467,E2 377.218} C_DIS
LIN {X 19.2203,Y 79.0728,Z 83,A 70.6869,B 24.8922,C -2.3966,E1 25.0379,E2 373.9479} C_DIS
LIN {X 15.6148,Y 79.8634,Z 83,A 73.7561,B 24.8908,C -2.4118,E1 25.0294,E2 370.8468} C_DIS
LIN {X 12.8326,Y 80.358,Z 83,A 76.2516,B 24.8894,C -2.4274,E1 25.0225,E2 368.3166} C_DIS
LIN {X 7.9301,Y 80.9891,Z 83,A 79.3267,B 24.8905,C -2.416,E1 25.014,E2 365.2708} C_DIS
LIN {X 4.5678,Y 81.2469,Z 83,A 81.5578,B 24.8908,C -2.4119,E1 25.0078,E2 363.0505} C_DIS
LIN {X 1.2634,Y 81.3654,Z 83,A 83.9099,B 24.8908,C -2.4123,E1 25.0013,E2 360.6978} C_DIS
LIN {X -2.2298,Y 81.3439,Z 83,A 86.8236,B 24.8896,C -2.4249,E1 24.993,E2 357.7541} C_DIS
LIN {X -6.3905,Y 81.1239,Z 83,A 90.6262,B 24.8874,C -2.4489,E1 24.9823,E2 353.8927} C_DIS
LIN {X -11.8512,Y 80.5086,Z 83,A 92.7716,B 24.8922,C -2.3968,E1 24.9767,E2 351.8695} C_DIS
LIN {X -17.5623,Y 79.4578,Z 83,A 97.141,B 24.8918,C -2.4015,E1 24.9647,E2 347.4844} C_DIS
LIN {X -20.8374,Y 78.6626,Z 83,A 99.7956,B 24.8913,C -2.4071,E1 24.9574,E2 344.8125} C_DIS
LIN {X -26.1546,Y 77.0577,Z 83,A 103.4743,B 24.8923,C -2.3962,E1 24.9477,E2 341.1535} C_DIS
LIN {X -29.1596,Y 75.9716,Z 83,A 106.1629,B 24.8914,C -2.4055,E1 24.9406,E2 338.4372} C_DIS
LIN {X -35.4689,Y 73.2389,Z 83,A 111.1755,B 24.8916,C -2.403,E1 24.9278,E2 333.4182} C_DIS
LIN {X -40.2988,Y 70.6966,Z 83,A 114.8612,B 24.8926,C -2.3921,E1 24.9188,E2 329.7479} C_DIS
LIN {X -43.8008,Y 68.5817,Z 83,A 117.3947,B 24.8939,C -2.3773,E1 24.9129,E2 327.2418} C_DIS
LIN {X -49.0036,Y 64.9661,Z 83,A 121.6807,B 24.8952,C -2.3636,E1 24.9031,E2 322.9738} C_DIS
LIN {X -53.0302,Y 61.7239,Z 83,A 125.3607,B 24.8958,C -2.3567,E1 24.8952,E2 319.2962} C_DIS
LIN {X -57.0477,Y 58.0304,Z 83,A 129.2237,B 24.8965,C -2.3484,E1 24.8873,E2 315.4375} C_DIS
LIN {X -60.68,Y 54.2205,Z 83,A 133.0017,B 24.8972,C -2.3411,E1 24.8801,E2 311.6602} C_DIS
LIN {X -64.0648,Y 50.1772,Z 83,A 137.0072,B 24.8973,C -2.3392,E1 24.8729,E2 307.6407} C_DIS
LIN {X -67.1084,Y 46.0283,Z 83,A 140.3882,B 24.8987,C -2.323,E1 24.8674,E2 304.2818} C_DIS
LIN {X -68.9649,Y 43.1947,Z 83,A 142.9392,B 24.8989,C -2.3208,E1 24.8636,E2 301.7234} C_DIS
LIN {X -70.5015,Y 40.6384,Z 83,A 145.6402,B 24.8981,C -2.3307,E1 24.8597,E2 298.9847} C_DIS
LIN {X -73.1098,Y 35.7363,Z 83,A 148.8446,B 24.9007,C -2.3006,E1 24.8557,E2 295.8349} C_DIS
LIN {X -74.898,Y 31.8163,Z 83,A 152.3455,B 24.9004,C -2.3038,E1 24.8517,E2 292.3072} C_DIS
LIN {X -76.506,Y 27.7271,Z 83,A 155.6497,B 24.9008,C -2.2999,E1 24.8484,E2 288.9937} C_DIS
LIN {X -77.9375,Y 23.4039,Z 83,A 158.8017,B 24.9017,C -2.2885,E1 24.8458,E2 285.8508} C_DIS
LIN {X -79.1418,Y 18.9374,Z 83,A 161.452,B 24.904,C -2.2625,E1 24.844,E2 283.2473} C_DIS
LIN {X -80.282,Y 13.2941,Z 83,A 166.2174,B 24.9035,C -2.2681,E1 24.8415,E2 278.4401} C_DIS
LIN {X -81.0163,Y 7.6357,Z 83,A 169.7442,B 24.9057,C -2.2425,E1 24.8404,E2 274.9535} C_DIS
LIN {X -81.3457,Y 2.2083,Z 83,A 174.5023,B 24.9046,C -2.2547,E1 24.8398,E2 270.1376} C_DIS
LIN {X -81.3566,Y -1.761,Z 83,A 176.4632,B 24.9072,C -2.2239,E1 24.8398,E2 268.2385} C_DIS
LIN {X -81.1813,Y -5.6053,Z 83,A 179.2932,B 24.9077,C -2.2184,E1 24.8403,E2 265.4044} C_DIS
LIN {X -80.8514,Y -9.2109,Z 83,A -177.8237,B 24.9077,C -2.2192,E1 24.8411,E2 262.5023} C_DIS
LIN {X -80.3493,Y -12.8887,Z 83,A -175.6306,B 24.9092,C -2.1999,E1 24.842,E2 260.3421} C_DIS
LIN {X -79.2871,Y -18.3163,Z 83,A -171.7331,B 24.9102,C -2.188,E1 24.8442,E2 256.45} C_DIS
LIN {X -78.4358,Y -21.6787,Z 83,A -169.0965,B 24.9104,C -2.1857,E1 24.8461,E2 253.8035} C_DIS
LIN {X -77.1917,Y -25.7571,Z 83,A -166.1623,B 24.9113,C -2.175,E1 24.8486,E2 250.878} C_DIS
LIN {X -76.2078,Y -28.5374,Z 83,A -164.0677,B 24.9117,C -2.1695,E1 24.8506,E2 248.7849} C_DIS
LIN {X -74.8001,Y -32.0474,Z 83,A -160.3434,B 24.91,C -2.1903,E1 24.8547,E2 244.9902} C_DIS
LIN {X -72.8405,Y -36.2797,Z 83,A -158.0485,B 24.9129,C -2.1546,E1 24.8574,E2 242.7681} C_DIS
LIN {X -69.5659,Y -42.2198,Z 83,A -153.3407,B 24.9141,C -2.14,E1 24.8639,E2 238.0705} C_DIS
LIN {X -68.347,Y -44.1664,Z 83,A -151.2969,B 24.9135,C -2.1473,E1 24.867,E2 235.9988} C_DIS
LIN {X -65.0693,Y -48.8663,Z 83,A -147.3708,B 24.9146,C -2.1345,E1 24.8734,E2 232.0843} C_DIS
LIN {X -63.3932,Y -51.0226,Z 83,A -144.6376,B 24.9131,C -2.1522,E1 24.8783,E2 229.2961} C_DIS
LIN {X -60.3899,Y -54.5439,Z 83,A -142.2385,B 24.9156,C -2.1212,E1 24.8826,E2 226.9601} C_DIS
LIN {X -58.6824,Y -56.3765,Z 83,A -140.4167,B 24.9158,C -2.119,E1 24.8861,E2 225.1357} C_DIS
LIN {X -53.8569,Y -61.0045,Z 83,A -135.8147,B 24.9168,C -2.1066,E1 24.8955,E2 220.5446} C_DIS
LIN {X -50.8618,Y -63.5235,Z 83,A -132.9819,B 24.917,C -2.1036,E1 24.9016,E2 217.7081} C_DIS
LIN {X -48.1598,Y -65.594,Z 83,A -130.9005,B 24.918,C -2.0907,E1 24.9062,E2 215.6499} C_DIS
LIN {X -45.558,Y -67.427,Z 83,A -127.6369,B 24.916,C -2.1158,E1 24.9139,E2 212.3156} C_DIS
LIN {X -42.1588,Y -69.603,Z 83,A -125.5546,B 24.9181,C -2.0901,E1 24.9187,E2 210.288} C_DIS
LIN {X -39.771,Y -70.9944,Z 83,A -123.1703,B 24.9173,C -2.0999,E1 24.9246,E2 207.8734} C_DIS
LIN {X -35.4349,Y -73.2553,Z 83,A -120.1912,B 24.9187,C -2.0824,E1 24.932,E2 204.9279} C_DIS
LIN {X -31.4984,Y -75.0319,Z 83,A -116.7909,B 24.9181,C -2.0895,E1 24.9407,E2 201.5029} C_DIS
LIN {X -27.43,Y -76.6143,Z 83,A -114.0395,B 24.9191,C -2.0774,E1 24.9479,E2 198.7745} C_DIS
LIN {X -22.3502,Y -78.2459,Z 83,A -109.6685,B 24.9179,C -2.0926,E1 24.9597,E2 194.3599} C_DIS
LIN {X -18.9466,Y -79.1396,Z 83,A -107.816,B 24.9194,C -2.073,E1 24.9646,E2 192.5515} C_DIS
LIN {X -15.8219,Y -79.8235,Z 83,A -105.1593,B 24.9186,C -2.0839,E1 24.9719,E2 189.8658} C_DIS
LIN {X -10.6312,Y -80.678,Z 83,A -101.8426,B 24.9195,C -2.0716,E1 24.981,E2 186.5755} C_DIS
LIN {X -7.175,Y -81.0589,Z 83,A -99.553,B 24.9199,C -2.0666,E1 24.9873,E2 184.2963} C_DIS
LIN {X -3.2559,Y -81.3104,Z 83,A -96.4914,B 24.9192,C -2.0756,E1 24.9959,E2 181.2125} C_DIS
LIN {X 0.5364,Y -81.3719,Z 83,A -94.0593,B 24.9197,C -2.0691,E1 25.0027,E2 178.796} C_DIS
Enddeposition()
LIN {X 0.5364,Y -81.3719,Z 83,A -94.0593,B 24.9197,C -2.0691,E1 25.0027,E2 178.796} C_DIS
Startdeposition()
$VEL.CP = VEL_PRINT
LIN {X -1.459,Y -80.4101,Z 83,A -96.3247,B 24.9204,C -2.0604,E1 24.9963,E2 181.0818} C_DIS
LIN {X -6.3323,Y -80.1737,Z 83,A -99.9399,B 24.9207,C -2.0562,E1 24.9862,E2 184.7081} C_DIS
LIN {X -9.1096,Y -79.9061,Z 83,A -102.0781,B 24.921,C -2.0521,E1 24.9802,E2 186.8573} C_DIS
LIN {X -12.4547,Y -79.4533,Z 83,A -105.0692,B 24.9223,C -2.0362,E1 24.9718,E2 189.8889} C_DIS
LIN {X -16.1423,Y -78.7867,Z 83,A -107.0076,B 24.9206,C -2.0578,E1 24.9667,E2 191.7781} C_DIS
LIN {X -19.6968,Y -77.9738,Z 83,A -109.8693,B 24.9211,C -2.0518,E1 24.9588,E2 194.6581} C_DIS
LIN {X -25.1867,Y -76.379,Z 83,A -113.7555,B 24.9204,C -2.0598,E1 24.9485,E2 198.5318} C_DIS
LIN {X -27.9847,Y -75.3988,Z 83,A -115.8087,B 24.9202,C -2.0633,E1 24.9431,E2 200.5808} C_DIS
LIN {X -33.3173,Y -73.1981,Z 83,A -119.9023,B 24.9198,C -2.068,E1 24.9326,E2 204.6726} C_DIS
LIN {X -36.5568,Y -71.6346,Z 83,A -123.3885,B 24.9215,C -2.0461,E1 24.9238,E2 208.2204} C_DIS
LIN {X -40.2826,Y -69.6081,Z 83,A -125.0166,B 24.9182,C -2.088,E1 24.92,E2 209.7534} C_DIS
LIN {X -43.2053,Y -67.8324,Z 83,A -128.2885,B 24.9197,C -2.0689,E1 24.9121,E2 213.081} C_DIS
LIN {X -47.1059,Y -65.1857,Z 83,A -131.352,B 24.9187,C -2.0823,E1 24.9051,E2 216.1231} C_DIS
LIN {X -50.0001,Y -62.9916,Z 83,A -133.9913,B 24.9184,C -2.0855,E1 24.8993,E2 218.7643} C_DIS
LIN {X -52.5318,Y -60.898,Z 83,A -136.3593,B 24.9181,C -2.0892,E1 24.8943,E2 221.1328} C_DIS
LIN {X -55.8419,Y -57.8758,Z 83,A -140.0471,B 24.9187,C -2.0826,E1 24.8867,E2 224.8514} C_DIS
LIN {X -58.1184,Y -55.5902,Z 83,A -141.5362,B 24.9166,C -2.1088,E1 24.8839,E2 226.2844} C_DIS
LIN {X -60.5161,Y -52.9691,Z 83,A -144.8444,B 24.9178,C -2.094,E1 24.8777,E2 229.6426} C_DIS
LIN {X -63.2866,Y -49.6267,Z 83,A -148.0289,B 24.9174,C -2.0989,E1 24.8721,E2 232.8304} C_DIS
LIN {X -65.2314,Y -47.0406,Z 83,A -149.4764,B 24.9152,C -2.1268,E1 24.8698,E2 234.2183} C_DIS
LIN {X -67.7729,Y -43.2987,Z 83,A -153.0085,B 24.9152,C -2.1268,E1 24.8643,E2 237.768} C_DIS
LIN {X -71.1723,Y -37.4489,Z 83,A -157.7024,B 24.9139,C -2.1429,E1 24.8578,E2 242.448} C_DIS
LIN {X -72.113,Y -35.6041,Z 83,A -159.5303,B 24.9143,C -2.1379,E1 24.8555,E2 244.2977} C_DIS
LIN {X -73.7897,Y -31.9848,Z 83,A -162.7735,B 24.9145,C -2.1357,E1 24.8518,E2 247.5639} C_DIS
LIN {X -75.0363,Y -28.9431,Z 83,A -164.6463,B 24.9129,C -2.1544,E1 24.85,E2 249.4027} C_DIS
LIN {X -76.1403,Y -25.8961,Z 83,A -167.246,B 24.9129,C -2.1538,E1 24.8476,E2 252.0187} C_DIS
LIN {X -77.3561,Y -21.999,Z 83,A -169.8193,B 24.9116,C -2.171,E1 24.8455,E2 254.5658} C_DIS
LIN {X -78.4112,Y -17.8787,Z 83,A -174.0413,B 24.9133,C -2.1504,E1 24.8428,E2 258.8617} C_DIS
LIN {X -79.3779,Y -12.9297,Z 83,A -176.2887,B 24.9096,C -2.1951,E1 24.8417,E2 261.0156} C_DIS
LIN {X -79.8418,Y -9.6574,Z 83,A -178.9971,B 24.9097,C -2.1936,E1 24.8407,E2 263.7439} C_DIS
LIN {X -80.2128,Y -5.8037,Z 83,A 177.9781,B 24.9096,C -2.1956,E1 24.84,E2 266.782} C_DIS
LIN {X -80.3945,Y -2.174,Z 83,A 175.4979,B 24.9087,C -2.2065,E1 24.8398,E2 269.251} C_DIS
LIN {X -80.3956,Y 2.1396,Z 83,A 171.9695,B 24.9088,C -2.205,E1 24.84,E2 272.8044} C_DIS
LIN {X -80.2194,Y 5.7326,Z 83,A 170.004,B 24.9069,C -2.228,E1 24.8403,E2 274.7267} C_DIS
LIN {X -79.9278,Y 8.9249,Z 83,A 166.8262,B 24.9081,C -2.2131,E1 24.8413,E2 277.9592} C_DIS
LIN {X -79.3295,Y 13.2192,Z 83,A 165.1577,B 24.9043,C -2.2584,E1 24.842,E2 279.5294} C_DIS
LIN {X -78.4241,Y 17.823,Z 83,A 161.2766,B 24.9046,C -2.2553,E1 24.8442,E2 283.4407} C_DIS
LIN {X -77.3264,Y 22.1037,Z 83,A 158.2922,B 24.9034,C -2.2693,E1 24.8463,E2 286.4092} C_DIS
LIN {X -76.8071,Y 23.845,Z 83,A 156.0341,B 24.9051,C -2.2492,E1 24.8482,E2 288.7282} C_DIS
LIN {X -75.5599,Y 27.543,Z 83,A 154.0567,B 24.9027,C -2.2778,E1 24.85,E2 290.6486} C_DIS
LIN {X -73.9238,Y 31.6769,Z 83,A 150.7588,B 24.9021,C -2.284,E1 24.8535,E2 293.9499} C_DIS
LIN {X -72.5166,Y 34.7744,Z 83,A 148.4827,B 24.9012,C -2.295,E1 24.8561,E2 296.2123} C_DIS
LIN {X -69.7202,Y 40.0875,Z 83,A 143.3067,B 24.9021,C -2.2847,E1 24.8631,E2 301.44} C_DIS
LIN {X -67.7049,Y 43.4047,Z 83,A 141.2333,B 24.8999,C -2.3099,E1 24.8662,E2 303.4639} C_DIS
LIN {X -65.4594,Y 46.7224,Z 83,A 138.016,B 24.9,C -2.3085,E1 24.8713,E2 306.7005} C_DIS
LIN {X -62.6774,Y 50.394,Z 83,A 134.4624,B 24.8999,C -2.3102,E1 24.8775,E2 310.2667} C_DIS
LIN {X -60.3978,Y 53.1045,Z 83,A 132.9695,B 24.897,C -2.343,E1 24.8801,E2 311.6882} C_DIS
LIN {X -57.3509,Y 56.3811,Z 83,A 129.6058,B 24.8967,C -2.3462,E1 24.8865,E2 315.0589} C_DIS
LIN {X -56.0515,Y 57.6726,Z 83,A 127.1198,B 24.8991,C -2.3189,E1 24.8917,E2 317.6202} C_DIS
LIN {X -52.8044,Y 60.66,Z 83,A 125.4208,B 24.8952,C -2.3634,E1 24.895,E2 319.22} C_DIS
LIN {X -49.8342,Y 63.1226,Z 83,A 122.2342,B 24.8957,C -2.3578,E1 24.9019,E2 322.4319} C_DIS
LIN {X -47.0052,Y 65.2569,Z 83,A 118.9553,B 24.897,C -2.3433,E1 24.9094,E2 325.7569} C_DIS
LIN {X -44.0949,Y 67.2577,Z 83,A 117.0088,B 24.8952,C -2.363,E1 24.9139,E2 327.663} C_DIS
LIN {X -39.6572,Y 69.9675,Z 83,A 113.1068,B 24.8951,C -2.3645,E1 24.9232,E2 331.5734} C_DIS
LIN {X -35.8778,Y 71.9773,Z 83,A 110.3227,B 24.894,C -2.3765,E1 24.9301,E2 334.3363} C_DIS
LIN {X -33.8007,Y 72.9757,Z 83,A 108.2402,B 24.8948,C -2.3673,E1 24.9354,E2 336.4461} C_DIS
LIN {X -27.1655,Y 75.6976,Z 83,A 103.5152,B 24.8933,C -2.3845,E1 24.9476,E2 341.1404} C_DIS
LIN {X -22.0564,Y 77.3398,Z 83,A 99.3119,B 24.8938,C -2.3785,E1 24.9589,E2 345.3651} C_DIS
LIN {X -17.5354,Y 78.4894,Z 83,A 95.1231,B 24.8957,C -2.3582,E1 24.9705,E2 349.6077} C_DIS
LIN {X -12.3706,Y 79.4663,Z 83,A 92.1597,B 24.8935,C -2.382,E1 24.9785,E2 352.5171} C_DIS
LIN {X -6.631,Y 80.1498,Z 83,A 88.8369,B 24.8913,C -2.4062,E1 24.9875,E2 355.7843} C_DIS
LIN {X -2.8811,Y 80.3718,Z 83,A 85.753,B 24.8923,C -2.3958,E1 24.9962,E2 358.894} C_DIS
LIN {X 3.5401,Y 80.3454,Z 83,A 81.3068,B 24.8919,C -2.4001,E1 25.0086,E2 363.3294} C_DIS
LIN {X 8.2264,Y 80.0017,Z 83,A 78.1314,B 24.8915,C -2.4048,E1 25.0174,E2 366.492} C_DIS
LIN {X 13.267,Y 79.3215,Z 83,A 74.4244,B 24.8918,C -2.4015,E1 25.0277,E2 370.2037} C_DIS
LIN {X 15.7153,Y 78.874,Z 83,A 71.9729,B 24.8936,C -2.3813,E1 25.0345,E2 372.7002} C_DIS
LIN {X 19.1339,Y 78.1141,Z 83,A 69.4426,B 24.8938,C -2.3789,E1 25.0414,E2 375.2325} C_DIS
LIN {X 22.322,Y 77.2646,Z 83,A 67.5985,B 24.8926,C -2.3919,E1 25.0462,E2 377.0427} C_DIS
LIN {X 25.5633,Y 76.2526,Z 83,A 65.5536,B 24.8918,C -2.4009,E1 25.0516,E2 379.0624} C_DIS
LIN {X 30.3787,Y 74.4651,Z 83,A 61.6996,B 24.8927,C -2.3917,E1 25.0617,E2 382.9299} C_DIS
LIN {X 34.1254,Y 72.8246,Z 83,A 58.1266,B 24.8947,C -2.369,E1 25.0709,E2 386.5478} C_DIS
LIN {X 37.0725,Y 71.3705,Z 83,A 56.3652,B 24.8934,C -2.3831,E1 25.0752,E2 388.2709} C_DIS
LIN {X 42.3541,Y 68.3677,Z 83,A 51.7041,B 24.8949,C -2.367,E1 25.0865,E2 392.9559} C_DIS
LIN {X 46.0086,Y 65.9631,Z 83,A 47.9165,B 24.8971,C -2.342,E1 25.0953,E2 396.79} C_DIS
LIN {X 49.7103,Y 63.2206,Z 83,A 45.6572,B 24.8949,C -2.3667,E1 25.1002,E2 398.9824} C_DIS
LIN {X 53.2063,Y 60.3066,Z 83,A 41.723,B 24.8973,C -2.3396,E1 25.1086,E2 402.9653} C_DIS
LIN {X 55.9434,Y 57.7779,Z 83,A 39.9281,B 24.8955,C -2.3603,E1 25.1121,E2 404.7039} C_DIS
LIN {X 58.3864,Y 55.3085,Z 83,A 37.1202,B 24.8968,C -2.3448,E1 25.1176,E2 407.5365} C_DIS
LIN {X 61.2805,Y 52.0829,Z 83,A 34.4276,B 24.8964,C -2.3499,E1 25.1225,E2 410.2047} C_DIS
LIN {X 63.7805,Y 48.9895,Z 83,A 30.8679,B 24.8989,C -2.3208,E1 25.1288,E2 413.8166} C_DIS
LIN {X 65.7542,Y 46.3093,Z 83,A 28.9984,B 24.8981,C -2.3304,E1 25.1317,E2 415.6543} C_DIS
LIN {X 67.6805,Y 43.4427,Z 83,A 26.0936,B 24.8998,C -2.3104,E1 25.1362,E2 418.5919} C_DIS
LIN {X 70.4078,Y 38.8691,Z 83,A 22.7867,B 24.8994,C -2.3154,E1 25.1408,E2 421.8698} C_DIS
LIN {X 73.1197,Y 33.4913,Z 83,A 18.5419,B 24.9003,C -2.305,E1 25.146,E2 426.1165} C_DIS
LIN {X 74.4416,Y 30.4364,Z 83,A 15.3559,B 24.9031,C -2.2727,E1 25.1495,E2 429.3611} C_DIS
LIN {X 75.9304,Y 26.5048,Z 83,A 13.2816,B 24.9014,C -2.2928,E1 25.1514,E2 431.3764} C_DIS
LIN {X 76.7957,Y 23.8817,Z 83,A 10.6208,B 24.9037,C -2.2651,E1 25.1536,E2 434.0874} C_DIS
LIN {X 77.7881,Y 20.4181,Z 83,A 9.052,B 24.9017,C -2.2889,E1 25.1547,E2 435.5912} C_DIS
LIN {X 78.8973,Y 15.5976,Z 83,A 5.2243,B 24.9035,C -2.2684,E1 25.1571,E2 439.445} C_DIS
LIN {X 79.5006,Y 12.1484,Z 83,A 2.2787,B 24.9053,C -2.2464,E1 25.1584,E2 442.4253} C_DIS
LIN {X 80.2067,Y 5.9189,Z 83,A -1.7365,B 24.9053,C -2.2466,E1 25.1595,E2 446.4162} C_DIS
LIN {X 80.3803,Y 2.6354,Z 83,A -3.5843,B 24.9046,C -2.255,E1 25.1597,E2 448.2332} C_DIS
LIN {X 80.4191,Y -0.9517,Z 83,A -7.2696,B 24.9083,C -2.2109,E1 25.1597,E2 452.0008} C_DIS
LIN {X 80.2857,Y -4.7122,Z 83,A -9.2444,B 24.9072,C -2.2247,E1 25.1594,E2 453.9311} C_DIS
LIN {X 80.0873,Y -7.3447,Z 83,A -12.0398,B 24.9101,C -2.1897,E1 25.1587,E2 456.7926} C_DIS
LIN {X 79.5427,Y -11.8766,Z 83,A -14.0454,B 24.9076,C -2.2189,E1 25.1579,E2 458.7175} C_DIS
LIN {X 78.5971,Y -17.0416,Z 83,A -17.9858,B 24.9092,C -2.2006,E1 25.1559,E2 462.6781} C_DIS
LIN {X 77.8891,Y -20.03,Z 83,A -20.0792,B 24.9095,C -2.1967,E1 25.1545,E2 464.7685} C_DIS
LIN {X 77.0722,Y -22.974,Z 83,A -22.8283,B 24.9115,C -2.1717,E1 25.1523,E2 467.5608} C_DIS
LIN {X 75.6045,Y -27.4208,Z 83,A -26.4412,B 24.9131,C -2.1527,E1 25.1489,E2 471.1984} C_DIS
LIN {X 74.1673,Y -31.0989,Z 83,A -28.4197,B 24.9116,C -2.1706,E1 25.1469,E2 473.1238} C_DIS
LIN {X 72.2902,Y -35.2457,Z 83,A -31.7117,B 24.9125,C -2.1593,E1 25.143,E2 476.4246} C_DIS
LIN {X 69.9096,Y -39.7579,Z 83,A -35.2431,B 24.9131,C -2.152,E1 25.1383,E2 479.9547} C_DIS
LIN {X 68.736,Y -41.7527,Z 83,A -37.8676,B 24.916,C -2.1167,E1 25.1344,E2 482.6493} C_DIS
LIN {X 66.3061,Y -45.5152,Z 83,A -39.8851,B 24.9137,C -2.1446,E1 25.1314,E2 484.5908} C_DIS
LIN {X 64.0252,Y -48.6704,Z 83,A -42.9165,B 24.915,C -2.129,E1 25.1263,E2 487.6446} C_DIS
LIN {X 61.3597,Y -51.9894,Z 83,A -46.1428,B 24.9161,C -2.115,E1 25.1205,E2 490.8889} C_DIS
LIN {X 59.3947,Y -54.2239,Z 83,A -48.2184,B 24.9164,C -2.1111,E1 25.1167,E2 492.9647} C_DIS
LIN {X 56.7388,Y -56.9976,Z 83,A -50.6792,B 24.9163,C -2.113,E1 25.1119,E2 495.4105} C_DIS
LIN {X 53.4632,Y -60.0805,Z 83,A -54.0106,B 24.9172,C -2.1016,E1 25.105,E2 498.7553} C_DIS
LIN {X 51.6407,Y -61.6543,Z 83,A -56.0433,B 24.9182,C -2.0879,E1 25.1006,E2 500.8124} C_DIS
LIN {X 47.4286,Y -64.9496,Z 83,A -59.4123,B 24.9178,C -2.0935,E1 25.0932,E2 504.156} C_DIS
LIN {X 43.1132,Y -67.892,Z 83,A -62.7643,B 24.9175,C -2.0976,E1 25.0855,E2 507.4872} C_DIS
LIN {X 38.8656,Y -70.4098,Z 83,A -66.3876,B 24.9182,C -2.0879,E1 25.0767,E2 511.1222} C_DIS
LIN {X 36.5042,Y -71.6615,Z 83,A -69.1844,B 24.9206,C -2.0577,E1 25.0696,E2 513.983} C_DIS
LIN {X 33.1986,Y -73.2516,Z 83,A -71.0991,B 24.9193,C -2.0747,E1 25.0648,E2 515.8525} C_DIS
LIN {X 29.9099,Y -74.6549,Z 83,A -73.6677,B 24.9196,C -2.0704,E1 25.0582,E2 518.4253} C_DIS
LIN {X 25.6184,Y -76.234,Z 83,A -76.8411,B 24.9197,C -2.0687,E1 25.0499,E2 521.5961} C_DIS
LIN {X 21.7517,Y -77.4262,Z 83,A -79.9078,B 24.9204,C -2.06,E1 25.0416,E2 524.6782} C_DIS
LIN {X 16.9973,Y -78.6068,Z 83,A -83.4173,B 24.9207,C -2.0561,E1 25.0321,E2 528.192} C_DIS
LIN {X 14.2438,Y -79.1519,Z 83,A -86.5008,B 24.9233,C -2.0229,E1 25.0234,E2 531.3509} C_DIS
LIN {X 8.8966,Y -79.9311,Z 83,A -88.8381,B 24.9201,C -2.0645,E1 25.0172,E2 533.5877} C_DIS
LIN {X 3.3517,Y -80.3535,Z 83,A -93.0307,B 24.9207,C -2.0559,E1 25.0055,E2 537.7987} C_DIS
LIN {X 0.5347,Y -80.4066,Z 83,A -94.7861,B 24.9202,C -2.0629,E1 25.0006,E2 539.5373} C_DIS
Enddeposition()
LIN {X 0.5347,Y -80.4066,Z 83,A -94.7861,B 24.9202,C -2.0629,E1 25.0006,E2 539.5373} C_DIS
Startdeposition()
$VEL.CP = VEL_PRINT
LIN {X 0.7409,Y -79.4681,Z 83,A -93.703,B 24.9168,C -2.1065,E1 25.0039,E2 538.3509} C_DIS
LIN {X 3.382,Y -79.3995,Z 83,A -91.4949,B 24.916,C -2.1161,E1 25.0101,E2 536.1206} C_DIS
LIN {X 9.1526,Y -78.9427,Z 83,A -87.3196,B 24.9158,C -2.1184,E1 25.0217,E2 531.9425} C_DIS
LIN {X 14.9563,Y -78.0515,Z 83,A -83.7896,B 24.9172,C -2.1006,E1 25.0313,E2 528.4583} C_DIS
LIN {X 19.5782,Y -77.0224,Z 83,A -80.2793,B 24.9168,C -2.1067,E1 25.0409,E2 524.9385} C_DIS
LIN {X 23.9557,Y -75.7762,Z 83,A -77.138,B 24.9168,C -2.1061,E1 25.0493,E2 521.804} C_DIS
LIN {X 27.9889,Y -74.3799,Z 83,A -72.9727,B 24.9138,C -2.1432,E1 25.0605,E2 517.5593} C_DIS
LIN {X 31.7938,Y -72.8346,Z 83,A -71.3712,B 24.9168,C -2.106,E1 25.0644,E2 516.0497} C_DIS
LIN {X 33.5013,Y -72.0651,Z 83,A -69.3208,B 24.915,C -2.1294,E1 25.0697,E2 513.9491} C_DIS
LIN {X 37.3353,Y -70.1564,Z 83,A -66.2737,B 24.9146,C -2.1333,E1 25.0772,E2 510.9013} C_DIS
LIN {X 42.1681,Y -67.3615,Z 83,A -62.9829,B 24.9159,C -2.118,E1 25.0851,E2 507.6567} C_DIS
LIN {X 46.3589,Y -64.5495,Z 83,A -58.8779,B 24.9141,C -2.1395,E1 25.0946,E2 503.5147} C_DIS
LIN {X 50.9724,Y -60.972,Z 83,A -54.8041,B 24.9138,C -2.1443,E1 25.1036,E2 499.4447} C_DIS
LIN {X 53.7556,Y -58.5325,Z 83,A -51.9392,B 24.9128,C -2.1566,E1 25.1095,E2 496.5622} C_DIS
LIN {X 56.2241,Y -56.1667,Z 83,A -48.8501,B 24.9107,C -2.1822,E1 25.1158,E2 493.4255} C_DIS
LIN {X 58.6762,Y -53.599,Z 83,A -47.1271,B 24.9123,C -2.1621,E1 25.1189,E2 491.7576} C_DIS
LIN {X 61.6914,Y -50.0989,Z 83,A -43.7301,B 24.9115,C -2.1728,E1 25.1251,E2 488.3509} C_DIS
LIN {X 65.3799,Y -45.1801,Z 83,A -39.9325,B 24.9121,C -2.1646,E1 25.1314,E2 484.5908} C_DIS
LIN {X 67.4714,Y -41.9922,Z 83,A -37.0662,B 24.9112,C -2.1759,E1 25.1358,E2 481.712} C_DIS
LIN {X 68.6715,Y -40.0012,Z 83,A -34.1998,B 24.9077,C -2.2186,E1 25.1399,E2 478.7594} C_DIS
LIN {X 70.3655,Y -36.9381,Z 83,A -32.4964,B 24.9092,C -2.1997,E1 25.1421,E2 477.1096} C_DIS
LIN {X 71.7003,Y -34.2756,Z 83,A -29.6871,B 24.9069,C -2.2273,E1 25.1456,E2 474.2502} C_DIS
LIN {X 73.0285,Y -31.349,Z 83,A -27.9133,B 24.9078,C -2.2168,E1 25.1475,E2 472.511} C_DIS
LIN {X 74.6576,Y -27.2389,Z 83,A -24.9268,B 24.9075,C -2.2201,E1 25.1505,E2 469.5333} C_DIS
LIN {X 75.5133,Y -24.7703,Z 83,A -22.701,B 24.9061,C -2.2369,E1 25.1525,E2 467.2804} C_DIS
LIN {X 77.3066,Y -18.4277,Z 83,A -17.5303,B 24.9037,C -2.2653,E1 25.1562,E2 462.0724} C_DIS
LIN {X 78.0231,Y -15.1039,Z 83,A -15.2645,B 24.9036,C -2.2671,E1 25.1574,E2 459.8156} C_DIS
LIN {X 78.9306,Y -9.2567,Z 83,A -11.0818,B 24.9026,C -2.278,E1 25.159,E2 455.632} C_DIS
LIN {X 79.2577,Y -5.8455,Z 83,A -8.572,B 24.9019,C -2.2871,E1 25.1596,E2 453.1155} C_DIS
LIN {X 79.4653,Y -1.0675,Z 83,A -5.5836,B 24.9022,C -2.2833,E1 25.1598,E2 450.1539} C_DIS
LIN {X 79.4273,Y 2.66,Z 83,A -3.1872,B 24.9022,C -2.2825,E1 25.1597,E2 447.7735} C_DIS
LIN {X 79.3108,Y 5.0605,Z 83,A -0.4524,B 24.899,C -2.3203,E1 25.1592,E2 444.9658} C_DIS
LIN {X 78.9704,Y 8.9167,Z 83,A 1.6296,B 24.9002,C -2.3062,E1 25.1586,E2 442.9295} C_DIS
LIN {X 78.4306,Y 12.8233,Z 83,A 4.3902,B 24.8997,C -2.3124,E1 25.1574,E2 440.1704} C_DIS
LIN {X 77.4749,Y 17.7021,Z 83,A 8.0369,B 24.8985,C -2.3254,E1 25.1553,E2 436.5142} C_DIS
LIN {X 76.0488,Y 23.0765,Z 83,A 11.8456,B 24.898,C -2.3311,E1 25.1525,E2 432.714} C_DIS
LIN {X 75.2337,Y 25.606,Z 83,A 13.7558,B 24.8976,C -2.3366,E1 25.1508,E2 430.8016} C_DIS
LIN {X 73.6037,Y 29.9702,Z 83,A 17.1677,B 24.8966,C -2.348,E1 25.1474,E2 427.3817} C_DIS
LIN {X 72.2543,Y 33.0949,Z 83,A 20.0963,B 24.8946,C -2.3699,E1 25.144,E2 424.4171} C_DIS
LIN {X 70.099,Y 37.4441,Z 83,A 22.8554,B 24.8958,C -2.3561,E1 25.1406,E2 421.7053} C_DIS
LIN {X 66.6901,Y 43.2235,Z 83,A 27.8518,B 24.8943,C -2.3738,E1 25.1334,E2 416.6927} C_DIS
LIN {X 64.9759,Y 45.7612,Z 83,A 31.1635,B 24.8906,C -2.414,E1 25.1279,E2 413.3021} C_DIS
LIN {X 62.1123,Y 49.5775,Z 83,A 33.1799,B 24.8939,C -2.3776,E1 25.1246,E2 411.3812} C_DIS
LIN {X 59.7803,Y 52.3646,Z 83,A 36.5846,B 24.8912,C -2.408,E1 25.1183,E2 407.9202} C_DIS
LIN {X 55.6082,Y 56.7764,Z 83,A 41.0171,B 24.8902,C -2.419,E1 25.1096,E2 403.4806} C_DIS
LIN {X 53.2751,Y 58.9713,Z 83,A 43.4092,B 24.8895,C -2.4261,E1 25.1046,E2 401.0812} C_DIS
LIN {X 50.6692,Y 61.224,Z 83,A 45.2831,B 24.8908,C -2.4121,E1 25.1007,E2 399.2477} C_DIS
LIN {X 48.0627,Y 63.2919,Z 83,A 47.9082,B 24.8898,C -2.4232,E1 25.0949,E2 396.6058} C_DIS
LIN {X 44.7816,Y 65.6536,Z 83,A 50.3547,B 24.8906,C -2.4139,E1 25.0894,E2 394.1898} C_DIS
LIN {X 42.2842,Y 67.289,Z 83,A 53.1832,B 24.8885,C -2.4377,E1 25.0826,E2 391.3142} C_DIS
LIN {X 37.361,Y 70.1428,Z 83,A 56.4935,B 24.8901,C -2.4195,E1 25.0747,E2 388.0567} C_DIS
LIN {X 34.3018,Y 71.6877,Z 83,A 59.5968,B 24.8881,C -2.4414,E1 25.0668,E2 384.9098} C_DIS
LIN {X 30.6544,Y 73.3217,Z 83,A 61.9247,B 24.8894,C -2.4281,E1 25.0609,E2 382.619} C_DIS
LIN {X 26.5625,Y 74.9014,Z 83,A 64.9156,B 24.8895,C -2.4261,E1 25.0531,E2 379.6395} C_DIS
LIN {X 23.0594,Y 76.054,Z 83,A 67.992,B 24.8882,C -2.4403,E1 25.0449,E2 376.5349} C_DIS
LIN {X 18.9551,Y 77.178,Z 83,A 70.8019,B 24.8887,C -2.4347,E1 25.0373,E2 373.7426} C_DIS
LIN {X 13.591,Y 78.3022,Z 83,A 74.7325,B 24.8887,C -2.4358,E1 25.0266,E2 369.8144} C_DIS
LIN {X 8.5278,Y 79.013,Z 83,A 78.2607,B 24.889,C -2.4321,E1 25.0169,E2 366.2979} C_DIS
LIN {X 3.7081,Y 79.3855,Z 83,A 81.7742,B 24.889,C -2.433,E1 25.0071,E2 362.784} C_DIS
LIN {X -0.9855,Y 79.4668,Z 83,A 85.2828,B 24.8886,C -2.4359,E1 24.9973,E2 359.2688} C_DIS
LIN {X -5.587,Y 79.2752,Z 83,A 88.6465,B 24.8886,C -2.4359,E1 24.9879,E2 355.9042} C_DIS
LIN {X -8.2604,Y 79.041,Z 83,A 91.6455,B 24.886,C -2.4649,E1 24.9794,E2 352.8348} C_DIS
LIN {X -12.4652,Y 78.4885,Z 83,A 93.5329,B 24.8892,C -2.4301,E1 24.9744,E2 351.0285} C_DIS
LIN {X -16.8915,Y 77.6556,Z 83,A 96.5666,B 24.8899,C -2.4217,E1 24.9661,E2 348.0115} C_DIS
LIN {X -20.4999,Y 76.7823,Z 83,A 99.7373,B 24.8889,C -2.4326,E1 24.9574,E2 344.8103} C_DIS
LIN {X -23.5525,Y 75.9013,Z 83,A 102.3155,B 24.8885,C -2.4379,E1 24.9505,E2 342.215} C_DIS
LIN {X -26.7537,Y 74.8343,Z 83,A 104.9146,B 24.8883,C -2.4394,E1 24.9436,E2 339.6073} C_DIS
LIN {X -31.0304,Y 73.1633,Z 83,A 107.6284,B 24.8902,C -2.4187,E1 24.9367,E2 336.9367} C_DIS
LIN {X -32.6853,Y 72.4389,Z 83,A 109.0536,B 24.8901,C -2.4201,E1 24.933,E2 335.5048} C_DIS
LIN {X -35.3792,Y 71.1621,Z 83,A 111.1728,B 24.8905,C -2.4159,E1 24.9277,E2 333.3901} C_DIS
LIN {X -39.2752,Y 69.0892,Z 83,A 114.3918,B 24.8909,C -2.4115,E1 24.9198,E2 330.1725} C_DIS
LIN {X -42.8586,Y 66.9243,Z 83,A 117.0192,B 24.8923,C -2.3957,E1 24.9137,E2 327.5747} C_DIS
LIN {X -44.9185,Y 65.5606,Z 83,A 119.4162,B 24.8911,C -2.4085,E1 24.908,E2 325.1393} C_DIS
LIN {X -48.0186,Y 63.325,Z 83,A 121.9635,B 24.8921,C -2.3973,E1 24.9023,E2 322.6095} C_DIS
LIN {X -50.1057,Y 61.6859,Z 83,A 124.2186,B 24.8917,C -2.4022,E1 24.8974,E2 320.3343} C_DIS
LIN {X -54.4266,Y 57.9091,Z 83,A 128.352,B 24.8926,C -2.3927,E1 24.8888,E2 316.2071} C_DIS
LIN {X -57.6728,Y 54.6773,Z 83,A 131.884,B 24.8927,C -2.3907,E1 24.8819,E2 312.6647} C_DIS
LIN {X -61.2698,Y 50.614,Z 83,A 135.3857,B 24.8946,C -2.3701,E1 24.8756,E2 309.1963} C_DIS
LIN {X -63.1075,Y 48.3035,Z 83,A 137.7389,B 24.8946,C -2.3702,E1 24.8715,E2 306.8315} C_DIS
LIN {X -65.8511,Y 44.4899,Z 83,A 140.4935,B 24.8968,C -2.3448,E1 24.8672,E2 304.124} C_DIS
LIN {X -67.042,Y 42.6753,Z 83,A 143.1219,B 24.8948,C -2.3678,E1 24.8631,E2 301.4276} C_DIS
LIN {X -68.7806,Y 39.8123,Z 83,A 144.8214,B 24.897,C -2.3425,E1 24.8608,E2 299.7796} C_DIS
LIN {X -70.9425,Y 35.8194,Z 83,A 148.31,B 24.8974,C -2.3384,E1 24.8562,E2 296.2821} C_DIS
LIN {X -72.2872,Y 33.0219,Z 83,A 150.5558,B 24.898,C -2.332,E1 24.8536,E2 294.0395} C_DIS
LIN {X -74.1786,Y 28.5205,Z 83,A 153.9145,B 24.8993,C -2.3173,E1 24.8501,E2 290.6973} C_DIS
LIN {X -75.9312,Y 23.456,Z 83,A 157.5993,B 24.9007,C -2.3008,E1 24.8468,E2 287.0308} C_DIS
LIN {X -76.921,Y 19.9728,Z 83,A 160.5287,B 24.9007,C -2.3007,E1 24.8446,E2 284.0846} C_DIS
LIN {X -77.5975,Y 17.158,Z 83,A 163.2493,B 24.8999,C -2.3102,E1 24.8429,E2 281.3253} C_DIS
LIN {X -78.2417,Y 13.9276,Z 83,A 164.7565,B 24.9024,C -2.2807,E1 24.8422,E2 279.8797} C_DIS
LIN {X -78.8537,Y 9.8951,Z 83,A 168.0844,B 24.9024,C -2.2811,E1 24.8408,E2 276.531} C_DIS
LIN {X -79.2063,Y 6.4884,Z 83,A 170.457,B 24.9033,C -2.2708,E1 24.8402,E2 274.1688} C_DIS
LIN {X -79.4452,Y 2.0749,Z 83,A 174.3373,B 24.9026,C -2.2783,E1 24.8398,E2 270.2473} C_DIS
LIN {X -79.4609,Y -1.3071,Z 83,A 176.1648,B 24.9046,C -2.2549,E1 24.8398,E2 268.4644} C_DIS
LIN {X -79.345,Y -4.4825,Z 83,A 179.1042,B 24.9038,C -2.2642,E1 24.8403,E2 265.4851} C_DIS
LIN {X -79.0757,Y -7.9296,Z 83,A -178.4152,B 24.9045,C -2.2561,E1 24.841,E2 263.0092} C_DIS
LIN {X -78.6774,Y -11.2065,Z 83,A -176.8528,B 24.9069,C -2.2278,E1 24.8415,E2 261.505} C_DIS
LIN {X -78.28,Y -13.7143,Z 83,A -173.9565,B 24.9051,C -2.2494,E1 24.843,E2 258.54} C_DIS
LIN {X -77.4973,Y -17.606,Z 83,A -172.2308,B 24.9083,C -2.2115,E1 24.8439,E2 256.8946} C_DIS
LIN {X -76.5896,Y -21.2125,Z 83,A -169.1078,B 24.908,C -2.2146,E1 24.8461,E2 253.7459} C_DIS
LIN {X -75.5826,Y -24.5562,Z 83,A -166.4486,B 24.9083,C -2.2108,E1 24.8484,E2 251.0805} C_DIS
LIN {X -74.2795,Y -28.2539,Z 83,A -163.003,B 24.9077,C -2.2186,E1 24.8518,E2 247.5969} C_DIS
LIN {X -72.7786,Y -31.9223,Z 83,A -161.1234,B 24.9104,C -2.1851,E1 24.8538,E2 245.7867} C_DIS
LIN {X -70.9651,Y -35.7753,Z 83,A -157.804,B 24.9106,C -2.183,E1 24.8578,E2 242.4544} C_DIS
LIN {X -69.3859,Y -38.7464,Z 83,A -154.7631,B 24.9098,C -2.1926,E1 24.862,E2 239.3746} C_DIS
LIN {X -67.6028,Y -41.7819,Z 83,A -153.1114,B 24.9123,C -2.1628,E1 24.8643,E2 237.7857} C_DIS
LIN {X -65.399,Y -45.1523,Z 83,A -149.9551,B 24.9123,C -2.162,E1 24.8692,E2 234.6153} C_DIS
LIN {X -62.6221,Y -48.9325,Z 83,A -146.7696,B 24.9134,C -2.1487,E1 24.8745,E2 231.4464} C_DIS
LIN {X -58.388,Y -53.9131,Z 83,A -142.0564,B 24.9143,C -2.1379,E1 24.8831,E2 226.7374} C_DIS
LIN {X -56.7952,Y -55.5892,Z 83,A -139.1092,B 24.9118,C -2.1687,E1 24.889,E2 223.7042} C_DIS
LIN {X -53.5245,Y -58.7446,Z 83,A -137.0347,B 24.9149,C -2.1297,E1 24.8931,E2 221.7142} C_DIS
LIN {X -51.5493,Y -60.4846,Z 83,A -134.92,B 24.9148,C -2.1319,E1 24.8975,E2 219.586} C_DIS
LIN {X -49.0025,Y -62.5667,Z 83,A -132.4095,B 24.9148,C -2.1314,E1 24.903,E2 217.0674} C_DIS
LIN {X -46.6079,Y -64.3708,Z 83,A -130.2591,B 24.9151,C -2.1274,E1 24.9079,E2 214.919} C_DIS
LIN {X -43.15,Y -66.7373,Z 83,A -127.0698,B 24.9151,C -2.1272,E1 24.9153,E2 211.7196} C_DIS
LIN {X -40.0243,Y -68.6586,Z 83,A -124.6062,B 24.9158,C -2.1184,E1 24.9212,E2 209.2694} C_DIS
LIN {X -35.998,Y -70.8512,Z 83,A -120.99,B 24.9155,C -2.1228,E1 24.9302,E2 205.6328} C_DIS
LIN {X -32.7131,Y -72.4264,Z 83,A -118.1387,B 24.9152,C -2.1261,E1 24.9375,E2 202.7665} C_DIS
LIN {X -29.5984,Y -73.7551,Z 83,A -116.1856,B 24.9165,C -2.11,E1 24.9424,E2 200.8474} C_DIS
LIN {X -25.8712,Y -75.144,Z 83,A -113.3453,B 24.9168,C -2.1067,E1 24.9499,E2 198.0092} C_DIS
LIN {X -21.9456,Y -76.3819,Z 83,A -110.6133,B 24.9175,C -2.098,E1 24.9571,E2 195.2933} C_DIS
LIN {X -16.789,Y -77.678,Z 83,A -107.2384,B 24.9186,C -2.083,E1 24.9662,E2 191.9493} C_DIS
LIN {X -11.8172,Y -78.5887,Z 83,A -103.2738,B 24.918,C -2.0907,E1 24.9772,E2 187.9623} C_DIS
LIN {X -7.5456,Y -79.1128,Z 83,A -100.0811,B 24.9179,C -2.0928,E1 24.986,E2 184.7626} C_DIS
LIN {X -1.9695,Y -79.4485,Z 83,A -95.4157,B 24.9164,C -2.1116,E1 24.9992,E2 180.0514} C_DIS
LIN {X -1.9695,Y -79.4485,Z 83,A -95.4157,B 24.9164,C -2.1116,E1 24.9992,E2 180.0514} C_DIS
Enddeposition()
LIN {X 0.5307,Y -78.5002,Z 83,A -94.3535,B 24.9167,C -2.1071,E1 25.0021,E2 178.9997} C_DIS
Startdeposition()
$VEL.CP = VEL_PRINT
LIN {X -2.0438,Y -78.4939,Z 83,A -97.6798,B 24.92,C -2.0657,E1 24.9925,E2 182.4247} C_DIS
LIN {X -5.5748,Y -78.322,Z 83,A -99.3996,B 24.9181,C -2.0896,E1 24.9879,E2 184.0884} C_DIS
LIN {X -10.7051,Y -77.7872,Z 83,A -103.1184,B 24.918,C -2.0913,E1 24.9776,E2 187.8054} C_DIS
LIN {X -14.2409,Y -77.2182,Z 83,A -106.0171,B 24.9185,C -2.0842,E1 24.9696,E2 190.7238} C_DIS
LIN {X -17.0736,Y -76.6417,Z 83,A -108.6585,B 24.9196,C -2.0706,E1 24.9623,E2 193.4008} C_DIS
LIN {X -20.2379,Y -75.8671,Z 83,A -110.438,B 24.9182,C -2.0882,E1 24.9575,E2 195.141} C_DIS
LIN {X -23.3737,Y -74.9601,Z 83,A -112.7256,B 24.9179,C -2.0925,E1 24.9514,E2 197.4224} C_DIS
LIN {X -26.4847,Y -73.9195,Z 83,A -115.2223,B 24.9179,C -2.0916,E1 24.9448,E2 199.9259} C_DIS
LIN {X -29.8782,Y -72.6128,Z 83,A -118.1561,B 24.9183,C -2.0867,E1 24.9372,E2 202.8778} C_DIS
LIN {X -32.5227,Y -71.4681,Z 83,A -120.5743,B 24.9188,C -2.0806,E1 24.931,E2 205.3164} C_DIS
LIN {X -35.4391,Y -70.0679,Z 83,A -122.3853,B 24.9175,C -2.098,E1 24.9265,E2 207.0907} C_DIS
LIN {X -38.2968,Y -68.547,Z 83,A -124.7972,B 24.9173,C -2.0999,E1 24.9206,E2 209.5051} C_DIS
LIN {X -42.5152,Y -66.0132,Z 83,A -128.7628,B 24.9177,C -2.0954,E1 24.9112,E2 213.4938} C_DIS
LIN {X -46.2073,Y -63.4844,Z 83,A -131.6876,B 24.9165,C -2.1096,E1 24.9045,E2 216.3948} C_DIS
LIN {X -49.0586,Y -61.3091,Z 83,A -134.3494,B 24.9163,C -2.1131,E1 24.8987,E2 219.058} C_DIS
LIN {X -51.7018,Y -59.0954,Z 83,A -136.7645,B 24.9157,C -2.1205,E1 24.8936,E2 221.4649} C_DIS
LIN {X -53.2927,Y -57.6654,Z 83,A -138.889,B 24.9166,C -2.1092,E1 24.8892,E2 223.6251} C_DIS
LIN {X -56.7166,Y -54.3013,Z 83,A -141.8578,B 24.9149,C -2.1302,E1 24.8834,E2 226.5564} C_DIS
LIN {X -58.2411,Y -52.6637,Z 83,A -143.9905,B 24.9156,C -2.121,E1 24.8793,E2 228.7204} C_DIS
LIN {X -61.2013,Y -49.1918,Z 83,A -146.7158,B 24.9138,C -2.1441,E1 24.8745,E2 231.4034} C_DIS
LIN {X -63.2282,Y -46.5572,Z 83,A -149.4423,B 24.9139,C -2.1423,E1 24.8699,E2 234.1471} C_DIS
LIN {X -65.5731,Y -43.1915,Z 83,A -152.3645,B 24.9132,C -2.1516,E1 24.8654,E2 237.0617} C_DIS
Enddeposition()
END
